LIN {X 0,Y 319.56,Z 711.312,A -85,B 0,C 180,E1 -15773.491,E2 -15773.491} C_VEL
LIN {X 0,Y 321.103,Z 700.055,A -85,B 0,C 180,E1 -15774.745,E2 -15774.745} C_VEL
LIN {X 0,Y 322.479,Z 688.391,A -85,B 0,C 180,E1 -15775.754,E2 -15775.754} C_VEL
LIN {X 0,Y 323.352,Z 677.795,A -85,B 0,C 180,E1 -15776.459,E2 -15776.459} C_VEL
LIN {X 0,Y 324.244,Z 665.597,A -85,B 0,C 180,E1 -15777.032,E2 -15777.032} C_VEL
LIN {X 0,Y 324.808,Z 650.654,A -85,B 0,C 180,E1 -15777.446,E2 -15777.446} C_VEL
LIN {X 0,Y 326.381,Z 586.086,A -85,B 0,C 180,E1 -15778.864,E2 -15778.864} C_VEL
LIN {X 0,Y 324.427,Z 577.286,A -85,B 0,C 180,E1 -15779.252,E2 -15779.252} C_VEL
LIN {X 0,Y 318.211,Z 562.488,A -85,B 0,C 180,E1 -15780.197,E2 -15780.197} C_VEL
LIN {X 0,Y 314.383,Z 553.731,A -85,B 0,C 180,E1 -15780.82,E2 -15780.82} C_VEL
LIN {X 0,Y 312.516,Z 545.559,A -85,B 0,C 180,E1 -15783.889,E2 -15783.889} C_VEL
LIN {X 0,Y 312.541,Z 545.551,A -85,B 0,C 180,E1 -15787.382,E2 -15787.382} C_VEL
LIN {X 0,Y 312.524,Z 545.556,A -85,B 0,C 180,E1 -15790.332,E2 -15790.332} C_VEL
LIN {X 0,Y 311.845,Z 545.642,A -85,B 0,C 180,E1 -15791.408,E2 -15791.408} C_VEL
LIN {X 0,Y 308.973,Z 545.997,A -85,B 0,C 180,E1 -15793.16,E2 -15793.16} C_VEL
LIN {X 0,Y 306.557,Z 546.301,A -85,B 0,C 180,E1 -15794.58,E2 -15794.58} C_VEL
LIN {X 0,Y 305.543,Z 546.423,A -85,B 0,C 180,E1 -15795.68,E2 -15795.68} C_VEL
LIN {X 0,Y 305.472,Z 546.432,A -85,B 0,C 180,E1 -15796.052,E2 -15796.052} C_VEL
LIN {X 0,Y 305.463,Z 546.425,A -85,B 0,C 180,E1 -15799.893,E2 -15799.893} C_VEL
LIN {X 0,Y 305.499,Z 546.428,A -85,B 0,C 180,E1 -15803.625,E2 -15803.625} C_VEL
LIN {X 0,Y 305.461,Z 546.432,A -85,B 0,C 180,E1 -15806.482,E2 -15806.482} C_VEL
LIN {X 0,Y 305.458,Z 546.428,A -85,B 0,C 180,E1 -15809.59,E2 -15809.59} C_VEL
LIN {X 0,Y 305.516,Z 546.425,A -85,B 0,C 180,E1 -15812.608,E2 -15812.608} C_VEL
LIN {X 0,Y 305.503,Z 546.429,A -85,B 0,C 180,E1 -15815.538,E2 -15815.538} C_VEL
LIN {X 0,Y 305.514,Z 546.427,A -85,B 0,C 180,E1 -15819.814,E2 -15819.814} C_VEL
LIN {X 0,Y 305.568,Z 546.415,A -85,B 0,C 180,E1 -15822.602,E2 -15822.602} C_VEL
LIN {X 0,Y 305.642,Z 546.411,A -85,B 0,C 180,E1 -15825.348,E2 -15825.348} C_VEL
LIN {X 0,Y 305.629,Z 546.413,A -85,B 0,C 180,E1 -15829.399,E2 -15829.399} C_VEL
LIN {X 0,Y 305.79,Z 546.386,A -85,B 0,C 180,E1 -15832.074,E2 -15832.074} C_VEL
LIN {X 0,Y 305.681,Z 546.41,A -85,B 0,C 180,E1 -15834.723,E2 -15834.723} C_VEL
LIN {X 0,Y 305.952,Z 546.367,A -85,B 0,C 180,E1 -15838.684,E2 -15838.684} C_VEL
LIN {X 0,Y 305.952,Z 546.372,A -85,B 0,C 180,E1 -15841.316,E2 -15841.316} C_VEL
LIN {X 0,Y 305.835,Z 546.389,A -85,B 0,C 180,E1 -15846.598,E2 -15846.598} C_VEL
LIN {X 0,Y 305.697,Z 546.4,A -85,B 0,C 180,E1 -15849.261,E2 -15849.261} C_VEL
LIN {X 0,Y 305.581,Z 546.409,A -85,B 0,C 180,E1 -15853.296,E2 -15853.296} C_VEL
LIN {X 0,Y 305.587,Z 546.419,A -85,B 0,C 180,E1 -15856.02,E2 -15856.02} C_VEL
LIN {X 0,Y 305.569,Z 546.418,A -85,B 0,C 180,E1 -15859.444,E2 -15859.444} C_VEL
LIN {X 0,Y 305.48,Z 546.426,A -85,B 0,C 180,E1 -15863.04,E2 -15863.04} C_VEL
LIN {X 0,Y 305.542,Z 546.423,A -85,B 0,C 180,E1 -15866.227,E2 -15866.227} C_VEL
LIN {X 0,Y 305.491,Z 546.431,A -85,B 0,C 180,E1 -15869.051,E2 -15869.051} C_VEL
LIN {X 0,Y 305.46,Z 546.434,A -85,B 0,C 180,E1 -15873.517,E2 -15873.517} C_VEL
LIN {X 0,Y 305.492,Z 546.434,A -85,B 0,C 180,E1 -15876.737,E2 -15876.737} C_VEL
LIN {X 0,Y 305.46,Z 546.438,A -85,B 0,C 180,E1 -15880.603,E2 -15880.603} C_VEL
LIN {X 0,Y 305.477,Z 546.434,A -85,B 0,C 180,E1 -15883.646,E2 -15883.646} C_VEL
LIN {X 0,Y 305.456,Z 546.437,A -85,B 0,C 180,E1 -15887.414,E2 -15887.414} C_VEL
LIN {X 0,Y 305.474,Z 546.435,A -85,B 0,C 180,E1 -15891.598,E2 -15891.598} C_VEL
LIN {X 0,Y 305.486,Z 546.463,A -85,B 0,C 180,E1 -15895.243,E2 -15895.243} C_VEL
LIN {X 0,Y 308.154,Z 557.631,A -85,B 0,C 180,E1 -15899.128,E2 -15899.128} C_VEL
LIN {X 0,Y 310.414,Z 568.645,A -85,B 0,C 180,E1 -15902.711,E2 -15902.711} C_VEL
LIN {X 0,Y 310.525,Z 569.174,A -85,B 0,C 180,E1 -15902.861,E2 -15902.861} C_VEL
LIN {X 0,Y 313.109,Z 576.135,A -85,B 0,C 180,E1 -15903.297,E2 -15903.297} C_VEL
LIN {X 0,Y 318.037,Z 602.027,A -85,B 0,C 180,E1 -15904.418,E2 -15904.418} C_VEL
LIN {X 0,Y 319.468,Z 612.293,A -85,B 0,C 180,E1 -15904.803,E2 -15904.803} C_VEL
LIN {X 0,Y 317.655,Z 677.964,A -85,B 0,C 180,E1 -15906.3,E2 -15906.3} C_VEL
LIN {X 0,Y 316.743,Z 691.271,A -85,B 0,C 180,E1 -15906.85,E2 -15906.85} C_VEL
LIN {X 0,Y 315.38,Z 704.306,A -85,B 0,C 180,E1 -15907.653,E2 -15907.653} C_VEL
LIN {X 0,Y 313.983,Z 716.101,A -85,B 0,C 180,E1 -15908.671,E2 -15908.671} C_VEL
LIN {X 0,Y 312.204,Z 727.465,A -85,B 0,C 180,E1 -15909.923,E2 -15909.923} C_VEL
LIN {X 0,Y 310.485,Z 737.722,A -85,B 0,C 180,E1 -15911.354,E2 -15911.354} C_VEL
LIN {X 0,Y 308.823,Z 747.523,A -85,B 0,C 180,E1 -15913.084,E2 -15913.084} C_VEL
LIN {X 0,Y 307.251,Z 756.594,A -85,B 0,C 180,E1 -15915.089,E2 -15915.089} C_VEL
LIN {X 0,Y 305.836,Z 763.695,A -85,B 0,C 180,E1 -15917.053,E2 -15917.053} C_VEL
LIN {X 0,Y 304.779,Z 770.182,A -85,B 0,C 180,E1 -15919.37,E2 -15919.37} C_VEL
LIN {X 0,Y 304.162,Z 774.48,A -85,B 0,C 180,E1 -15921.362,E2 -15921.362} C_VEL
LIN {X 0,Y 303.743,Z 777.719,A -85,B 0,C 180,E1 -15923.357,E2 -15923.357} C_VEL
LIN {X 0,Y 303.631,Z 780.557,A -85,B 0,C 180,E1 -15926.018,E2 -15926.018} C_VEL
LIN {X 0,Y 303.606,Z 781.339,A -85,B 0,C 180,E1 -15927.347,E2 -15927.347} C_VEL
LIN {X 0,Y 303.605,Z 781.714,A -85,B 0,C 180,E1 -15930,E2 -15930} C_VEL
LIN {X 0,Y 303.575,Z 781.323,A -85,B 0,C 180,E1 -15931.327,E2 -15931.327} C_VEL
LIN {X 0,Y 303.608,Z 780.508,A -85,B 0,C 180,E1 -15932.653,E2 -15932.653} C_VEL
LIN {X 0,Y 303.631,Z 779.27,A -85,B 0,C 180,E1 -15933.982,E2 -15933.982} C_VEL
LIN {X 0,Y 303.66,Z 777.217,A -85,B 0,C 180,E1 -15935.611,E2 -15935.611} C_VEL
LIN {X 0,Y 303.953,Z 772.983,A -85,B 0,C 180,E1 -15937.974,E2 -15937.974} C_VEL
LIN {X 0,Y 304.414,Z 768.207,A -85,B 0,C 180,E1 -15939.971,E2 -15939.971} C_VEL
LIN {X 0,Y 305.31,Z 761.043,A -85,B 0,C 180,E1 -15942.294,E2 -15942.294} C_VEL
LIN {X 0,Y 306.496,Z 753.237,A -85,B 0,C 180,E1 -15944.27,E2 -15944.27} C_VEL
LIN {X 0,Y 307.813,Z 743.859,A -85,B 0,C 180,E1 -15946.165,E2 -15946.165} C_VEL
LIN {X 0,Y 309.152,Z 733.316,A -85,B 0,C 180,E1 -15947.872,E2 -15947.872} C_VEL
LIN {X 0,Y 310.628,Z 721.827,A -85,B 0,C 180,E1 -15949.322,E2 -15949.322} C_VEL
LIN {X 0,Y 311.964,Z 710.545,A -85,B 0,C 180,E1 -15950.437,E2 -15950.437} C_VEL
LIN {X 0,Y 313.093,Z 699.088,A -85,B 0,C 180,E1 -15951.306,E2 -15951.306} C_VEL
LIN {X 0,Y 314.068,Z 685.985,A -85,B 0,C 180,E1 -15952.013,E2 -15952.013} C_VEL
LIN {X 0,Y 314.673,Z 672.398,A -85,B 0,C 180,E1 -15952.472,E2 -15952.472} C_VEL
LIN {X 0,Y 316.012,Z 609.471,A -85,B 0,C 180,E1 -15953.888,E2 -15953.888} C_VEL
LIN {X 0,Y 311.128,Z 577.16,A -85,B 0,C 180,E1 -15955.044,E2 -15955.044} C_VEL
LIN {X 0,Y 309.749,Z 569.178,A -85,B 0,C 180,E1 -15955.394,E2 -15955.394} C_VEL
LIN {X 0,Y 309.315,Z 564.88,A -85,B 0,C 180,E1 -15956.662,E2 -15956.662} C_VEL
LIN {X 0,Y 307.408,Z 555.133,A -85,B 0,C 180,E1 -15959.685,E2 -15959.685} C_VEL
LIN {X 0,Y 305.487,Z 546.434,A -85,B 0,C 180,E1 -15962.531,E2 -15962.531} C_VEL
LIN {X 0,Y 305.494,Z 546.43,A -85,B 0,C 180,E1 -15966.736,E2 -15966.736} C_VEL
LIN {X 0,Y 305.452,Z 546.434,A -85,B 0,C 180,E1 -15970.599,E2 -15970.599} C_VEL
LIN {X 0,Y 305.424,Z 546.437,A -85,B 0,C 180,E1 -15974.493,E2 -15974.493} C_VEL
LIN {X 0,Y 305.475,Z 546.432,A -85,B 0,C 180,E1 -15978.149,E2 -15978.149} C_VEL
LIN {X 0,Y 305.504,Z 546.431,A -85,B 0,C 180,E1 -15981.602,E2 -15981.602} C_VEL
LIN {X 0,Y 305.457,Z 546.434,A -85,B 0,C 180,E1 -15984.886,E2 -15984.886} C_VEL
LIN {X 0,Y 305.446,Z 546.434,A -85,B 0,C 180,E1 -15988.355,E2 -15988.355} C_VEL
LIN {X 0,Y 305.515,Z 546.428,A -85,B 0,C 180,E1 -15991.113,E2 -15991.113} C_VEL
LIN {X 0,Y 305.565,Z 546.42,A -85,B 0,C 180,E1 -15994.087,E2 -15994.087} C_VEL
LIN {X 0,Y 305.475,Z 546.43,A -85,B 0,C 180,E1 -15998.401,E2 -15998.401} C_VEL
LIN {X 0,Y 305.573,Z 546.422,A -85,B 0,C 180,E1 -16001.217,E2 -16001.217} C_VEL
LIN {X 0,Y 305.642,Z 546.414,A -85,B 0,C 180,E1 -16005.349,E2 -16005.349} C_VEL
LIN {X 0,Y 305.631,Z 546.412,A -85,B 0,C 180,E1 -16009.4,E2 -16009.4} C_VEL
LIN {X 0,Y 305.802,Z 546.391,A -85,B 0,C 180,E1 -16012.074,E2 -16012.074} C_VEL
LIN {X 0,Y 305.681,Z 546.403,A -85,B 0,C 180,E1 -16014.723,E2 -16014.723} C_VEL
LIN {X 0,Y 305.95,Z 546.372,A -85,B 0,C 180,E1 -16018.684,E2 -16018.684} C_VEL
LIN {X 0,Y 305.95,Z 546.374,A -85,B 0,C 180,E1 -16021.316,E2 -16021.316} C_VEL
LIN {X 0,Y 305.682,Z 546.408,A -85,B 0,C 180,E1 -16025.277,E2 -16025.277} C_VEL
LIN {X 0,Y 305.79,Z 546.391,A -85,B 0,C 180,E1 -16027.926,E2 -16027.926} C_VEL
LIN {X 0,Y 305.596,Z 546.413,A -85,B 0,C 180,E1 -16031.946,E2 -16031.946} C_VEL
LIN {X 0,Y 305.631,Z 546.413,A -85,B 0,C 180,E1 -16035.035,E2 -16035.035} C_VEL
LIN {X 0,Y 305.57,Z 546.417,A -85,B 0,C 180,E1 -16039.445,E2 -16039.445} C_VEL
LIN {X 0,Y 305.485,Z 546.431,A -85,B 0,C 180,E1 -16043.042,E2 -16043.042} C_VEL
LIN {X 0,Y 305.543,Z 546.421,A -85,B 0,C 180,E1 -16046.228,E2 -16046.228} C_VEL
LIN {X 0,Y 305.491,Z 546.431,A -85,B 0,C 180,E1 -16049.051,E2 -16049.051} C_VEL
LIN {X 0,Y 305.461,Z 546.437,A -85,B 0,C 180,E1 -16053.518,E2 -16053.518} C_VEL
LIN {X 0,Y 305.493,Z 546.426,A -85,B 0,C 180,E1 -16056.737,E2 -16056.737} C_VEL
LIN {X 0,Y 305.452,Z 546.434,A -85,B 0,C 180,E1 -16060.601,E2 -16060.601} C_VEL
LIN {X 0,Y 305.468,Z 546.435,A -85,B 0,C 180,E1 -16063.648,E2 -16063.648} C_VEL
LIN {X 0,Y 305.507,Z 546.432,A -85,B 0,C 180,E1 -16067.404,E2 -16067.404} C_VEL
LIN {X 0,Y 305.519,Z 546.429,A -85,B 0,C 180,E1 -16071.605,E2 -16071.605} C_VEL
LIN {X 0,Y 305.462,Z 546.434,A -85,B 0,C 180,E1 -16074.888,E2 -16074.888} C_VEL
LIN {X 0,Y 305.452,Z 546.435,A -85,B 0,C 180,E1 -16078.356,E2 -16078.356} C_VEL
LIN {X 0,Y 305.521,Z 546.431,A -85,B 0,C 180,E1 -16081.115,E2 -16081.115} C_VEL
LIN {X 0,Y 305.574,Z 546.419,A -85,B 0,C 180,E1 -16084.089,E2 -16084.089} C_VEL
LIN {X 0,Y 305.566,Z 546.631,A -85,B 0,C 180,E1 -16085.98,E2 -16085.98} C_VEL
LIN {X 0,Y 307.028,Z 553.759,A -85,B 0,C 180,E1 -16088.494,E2 -16088.494} C_VEL
LIN {X 0,Y 314.277,Z 572.979,A -85,B 0,C 180,E1 -16089.556,E2 -16089.556} C_VEL
LIN {X 0,Y 316.555,Z 584.974,A -85,B 0,C 180,E1 -16090.02,E2 -16090.02} C_VEL
LIN {X 0,Y 314.853,Z 660.952,A -85,B 0,C 180,E1 -16091.757,E2 -16091.757} C_VEL
LIN {X 0,Y 314.205,Z 673.84,A -85,B 0,C 180,E1 -16092.299,E2 -16092.299} C_VEL
LIN {X 0,Y 313.3,Z 685.911,A -85,B 0,C 180,E1 -16093.046,E2 -16093.046} C_VEL
LIN {X 0,Y 312.168,Z 697.305,A -85,B 0,C 180,E1 -16093.991,E2 -16093.991} C_VEL
LIN {X 0,Y 310.905,Z 708.975,A -85,B 0,C 180,E1 -16095.268,E2 -16095.268} C_VEL
LIN {X 0,Y 309.493,Z 719.45,A -85,B 0,C 180,E1 -16096.708,E2 -16096.708} C_VEL
LIN {X 0,Y 308.138,Z 728.021,A -85,B 0,C 180,E1 -16098.155,E2 -16098.155} C_VEL
LIN {X 0,Y 307.155,Z 735.978,A -85,B 0,C 180,E1 -16099.805,E2 -16099.805} C_VEL
LIN {X 0,Y 306.074,Z 743.623,A -85,B 0,C 180,E1 -16101.749,E2 -16101.749} C_VEL
LIN {X 0,Y 305.32,Z 748.885,A -85,B 0,C 180,E1 -16103.391,E2 -16103.391} C_VEL
LIN {X 0,Y 304.67,Z 754.01,A -85,B 0,C 180,E1 -16105.369,E2 -16105.369} C_VEL
LIN {X 0,Y 303.991,Z 758.003,A -85,B 0,C 180,E1 -16107.35,E2 -16107.35} C_VEL
LIN {X 0,Y 303.805,Z 760.064,A -85,B 0,C 180,E1 -16108.674,E2 -16108.674} C_VEL
LIN {X 0,Y 303.616,Z 762.942,A -85,B 0,C 180,E1 -16111.326,E2 -16111.326} C_VEL
LIN {X 0,Y 303.632,Z 763.785,A -85,B 0,C 180,E1 -16112.653,E2 -16112.653} C_VEL
LIN {X 0,Y 303.647,Z 764.2,A -85,B 0,C 180,E1 -16113.981,E2 -16113.981} C_VEL
LIN {X 0,Y 303.697,Z 764.191,A -85,B 0,C 180,E1 -16115.678,E2 -16115.678} C_VEL
LIN {X 0,Y 303.777,Z 763.154,A -85,B 0,C 180,E1 -16117.979,E2 -16117.979} C_VEL
LIN {X 0,Y 303.939,Z 761.978,A -85,B 0,C 180,E1 -16119.315,E2 -16119.315} C_VEL
LIN {X 0,Y 304.161,Z 760.397,A -85,B 0,C 180,E1 -16120.652,E2 -16120.652} C_VEL
LIN {X 0,Y 304.752,Z 757.208,A -85,B 0,C 180,E1 -16122.655,E2 -16122.655} C_VEL
LIN {X 0,Y 305.742,Z 751.858,A -85,B 0,C 180,E1 -16125.105,E2 -16125.105} C_VEL
LIN {X 0,Y 306.938,Z 745.372,A -85,B 0,C 180,E1 -16127.317,E2 -16127.317} C_VEL
LIN {X 0,Y 308.349,Z 737.987,A -85,B 0,C 180,E1 -16129.298,E2 -16129.298} C_VEL
LIN {X 0,Y 309.874,Z 730.443,A -85,B 0,C 180,E1 -16130.929,E2 -16130.929} C_VEL
LIN {X 0,Y 311.396,Z 721.288,A -85,B 0,C 180,E1 -16132.561,E2 -16132.561} C_VEL
LIN {X 0,Y 313.002,Z 711.086,A -85,B 0,C 180,E1 -16134.014,E2 -16134.014} C_VEL
LIN {X 0,Y 314.624,Z 699.733,A -85,B 0,C 180,E1 -16135.29,E2 -16135.29} C_VEL
LIN {X 0,Y 316.05,Z 687.935,A -85,B 0,C 180,E1 -16136.317,E2 -16136.317} C_VEL
LIN {X 0,Y 316.984,Z 677.136,A -85,B 0,C 180,E1 -16137.033,E2 -16137.033} C_VEL
LIN {X 0,Y 317.861,Z 664.324,A -85,B 0,C 180,E1 -16137.621,E2 -16137.621} C_VEL
LIN {X 0,Y 318.495,Z 646.755,A -85,B 0,C 180,E1 -16138.08,E2 -16138.08} C_VEL
LIN {X 0,Y 319.984,Z 586.641,A -85,B 0,C 180,E1 -16139.429,E2 -16139.429} C_VEL
LIN {X 0,Y 318.28,Z 579.564,A -85,B 0,C 180,E1 -16139.764,E2 -16139.764} C_VEL
LIN {X 0,Y 311.901,Z 564.373,A -85,B 0,C 180,E1 -16140.769,E2 -16140.769} C_VEL
LIN {X 0,Y 307.227,Z 553.981,A -85,B 0,C 180,E1 -16141.541,E2 -16141.541} C_VEL
LIN {X 0,Y 305.461,Z 546.438,A -85,B 0,C 180,E1 -16144.464,E2 -16144.464} C_VEL
LIN {X 0,Y 305.509,Z 546.427,A -85,B 0,C 180,E1 -16148.396,E2 -16148.396} C_VEL
LIN {X 0,Y 305.507,Z 546.432,A -85,B 0,C 180,E1 -16152.596,E2 -16152.596} C_VEL
LIN {X 0,Y 305.472,Z 546.432,A -85,B 0,C 180,E1 -16156.052,E2 -16156.052} C_VEL
LIN {X 0,Y 304.825,Z 546.516,A -85,B 0,C 180,E1 -16157.152,E2 -16157.152} C_VEL
LIN {X 0,Y 301.953,Z 546.873,A -85,B 0,C 180,E1 -16158.94,E2 -16158.94} C_VEL
LIN {X 0,Y 299.517,Z 547.173,A -85,B 0,C 180,E1 -16160.392,E2 -16160.392} C_VEL
LIN {X 0,Y 298.495,Z 547.303,A -85,B 0,C 180,E1 -16161.517,E2 -16161.517} C_VEL
LIN {X 0,Y 298.425,Z 547.31,A -85,B 0,C 180,E1 -16161.898,E2 -16161.898} C_VEL
LIN {X 0,Y 298.404,Z 547.311,A -85,B 0,C 180,E1 -16165.58,E2 -16165.58} C_VEL
LIN {X 0,Y 298.391,Z 547.313,A -85,B 0,C 180,E1 -16168.79,E2 -16168.79} C_VEL
LIN {X 0,Y 298.459,Z 547.307,A -85,B 0,C 180,E1 -16171.904,E2 -16171.904} C_VEL
LIN {X 0,Y 298.48,Z 547.306,A -85,B 0,C 180,E1 -16174.923,E2 -16174.923} C_VEL
LIN {X 0,Y 298.445,Z 547.309,A -85,B 0,C 180,E1 -16179.315,E2 -16179.315} C_VEL
LIN {X 0,Y 298.531,Z 547.291,A -85,B 0,C 180,E1 -16182.179,E2 -16182.179} C_VEL
LIN {X 0,Y 298.587,Z 547.291,A -85,B 0,C 180,E1 -16184.994,E2 -16184.994} C_VEL
LIN {X 0,Y 298.585,Z 547.292,A -85,B 0,C 180,E1 -16189.146,E2 -16189.146} C_VEL
LIN {X 0,Y 298.734,Z 547.266,A -85,B 0,C 180,E1 -16191.885,E2 -16191.885} C_VEL
LIN {X 0,Y 298.652,Z 547.284,A -85,B 0,C 180,E1 -16194.599,E2 -16194.599} C_VEL
LIN {X 0,Y 298.918,Z 547.242,A -85,B 0,C 180,E1 -16198.653,E2 -16198.653} C_VEL
LIN {X 0,Y 298.918,Z 547.248,A -85,B 0,C 180,E1 -16201.347,E2 -16201.347} C_VEL
LIN {X 0,Y 298.78,Z 547.266,A -85,B 0,C 180,E1 -16206.754,E2 -16206.754} C_VEL
LIN {X 0,Y 298.629,Z 547.281,A -85,B 0,C 180,E1 -16209.482,E2 -16209.482} C_VEL
LIN {X 0,Y 298.545,Z 547.285,A -85,B 0,C 180,E1 -16213.616,E2 -16213.616} C_VEL
LIN {X 0,Y 298.542,Z 547.299,A -85,B 0,C 180,E1 -16216.409,E2 -16216.409} C_VEL
LIN {X 0,Y 298.504,Z 547.298,A -85,B 0,C 180,E1 -16219.654,E2 -16219.654} C_VEL
LIN {X 0,Y 298.423,Z 547.306,A -85,B 0,C 180,E1 -16223.601,E2 -16223.601} C_VEL
LIN {X 0,Y 298.484,Z 547.299,A -85,B 0,C 180,E1 -16226.575,E2 -16226.575} C_VEL
LIN {X 0,Y 298.416,Z 547.311,A -85,B 0,C 180,E1 -16229.641,E2 -16229.641} C_VEL
LIN {X 0,Y 298.39,Z 547.317,A -85,B 0,C 180,E1 -16232.801,E2 -16232.801} C_VEL
LIN {X 0,Y 298.461,Z 547.309,A -85,B 0,C 180,E1 -16236.813,E2 -16236.813} C_VEL
LIN {X 0,Y 298.415,Z 547.314,A -85,B 0,C 180,E1 -16241.095,E2 -16241.095} C_VEL
LIN {X 0,Y 298.385,Z 547.319,A -85,B 0,C 180,E1 -16244.959,E2 -16244.959} C_VEL
LIN {X 0,Y 298.385,Z 547.319,A -85,B 0,C 180,E1 -16248.913,E2 -16248.913} C_VEL
LIN {X 0,Y 298.444,Z 547.31,A -85,B 0,C 180,E1 -16253.193,E2 -16253.193} C_VEL
LIN {X 0,Y 298.467,Z 547.491,A -85,B 0,C 180,E1 -16254.661,E2 -16254.661} C_VEL
LIN {X 0,Y 301.166,Z 558.807,A -85,B 0,C 180,E1 -16258.721,E2 -16258.721} C_VEL
LIN {X 0,Y 303.324,Z 569.024,A -85,B 0,C 180,E1 -16262.11,E2 -16262.11} C_VEL
LIN {X 0,Y 307.136,Z 578.741,A -85,B 0,C 180,E1 -16262.765,E2 -16262.765} C_VEL
LIN {X 0,Y 311.765,Z 603.378,A -85,B 0,C 180,E1 -16263.861,E2 -16263.861} C_VEL
LIN {X 0,Y 313.119,Z 613.122,A -85,B 0,C 180,E1 -16264.238,E2 -16264.238} C_VEL
LIN {X 0,Y 311.298,Z 677.056,A -85,B 0,C 180,E1 -16265.715,E2 -16265.715} C_VEL
LIN {X 0,Y 310.396,Z 690.278,A -85,B 0,C 180,E1 -16266.26,E2 -16266.26} C_VEL
LIN {X 0,Y 309.097,Z 702.433,A -85,B 0,C 180,E1 -16266.997,E2 -16266.997} C_VEL
LIN {X 0,Y 307.628,Z 714.698,A -85,B 0,C 180,E1 -16268.032,E2 -16268.032} C_VEL
LIN {X 0,Y 305.781,Z 726.28,A -85,B 0,C 180,E1 -16269.307,E2 -16269.307} C_VEL
LIN {X 0,Y 303.959,Z 736.711,A -85,B 0,C 180,E1 -16270.763,E2 -16270.763} C_VEL
LIN {X 0,Y 302.138,Z 746.571,A -85,B 0,C 180,E1 -16272.496,E2 -16272.496} C_VEL
LIN {X 0,Y 300.619,Z 755.195,A -85,B 0,C 180,E1 -16274.404,E2 -16274.404} C_VEL
LIN {X 0,Y 299.147,Z 762.523,A -85,B 0,C 180,E1 -16276.413,E2 -16276.413} C_VEL
LIN {X 0,Y 298.083,Z 768.412,A -85,B 0,C 180,E1 -16278.44,E2 -16278.44} C_VEL
LIN {X 0,Y 297.302,Z 773.065,A -85,B 0,C 180,E1 -16280.475,E2 -16280.475} C_VEL
LIN {X 0,Y 296.804,Z 776.619,A -85,B 0,C 180,E1 -16282.517,E2 -16282.517} C_VEL
LIN {X 0,Y 296.552,Z 779.176,A -85,B 0,C 180,E1 -16284.561,E2 -16284.561} C_VEL
LIN {X 0,Y 296.528,Z 780.382,A -85,B 0,C 180,E1 -16285.923,E2 -16285.923} C_VEL
LIN {X 0,Y 296.533,Z 781.148,A -85,B 0,C 180,E1 -16287.283,E2 -16287.283} C_VEL
LIN {X 0,Y 296.52,Z 781.505,A -85,B 0,C 180,E1 -16290,E2 -16290} C_VEL
LIN {X 0,Y 296.494,Z 781.104,A -85,B 0,C 180,E1 -16291.358,E2 -16291.358} C_VEL
LIN {X 0,Y 296.534,Z 780.27,A -85,B 0,C 180,E1 -16292.717,E2 -16292.717} C_VEL
LIN {X 0,Y 296.529,Z 779.022,A -85,B 0,C 180,E1 -16294.077,E2 -16294.077} C_VEL
LIN {X 0,Y 296.553,Z 777.257,A -85,B 0,C 180,E1 -16295.522,E2 -16295.522} C_VEL
LIN {X 0,Y 296.786,Z 774.037,A -85,B 0,C 180,E1 -16297.483,E2 -16297.483} C_VEL
LIN {X 0,Y 297.214,Z 769.628,A -85,B 0,C 180,E1 -16299.527,E2 -16299.527} C_VEL
LIN {X 0,Y 297.873,Z 764.015,A -85,B 0,C 180,E1 -16301.569,E2 -16301.569} C_VEL
LIN {X 0,Y 298.899,Z 757.005,A -85,B 0,C 180,E1 -16303.599,E2 -16303.599} C_VEL
LIN {X 0,Y 300.253,Z 748.214,A -85,B 0,C 180,E1 -16305.615,E2 -16305.615} C_VEL
LIN {X 0,Y 301.512,Z 739.161,A -85,B 0,C 180,E1 -16307.296,E2 -16307.296} C_VEL
LIN {X 0,Y 302.862,Z 729.288,A -85,B 0,C 180,E1 -16308.782,E2 -16308.782} C_VEL
LIN {X 0,Y 304.321,Z 718.323,A -85,B 0,C 180,E1 -16310.091,E2 -16310.091} C_VEL
LIN {X 0,Y 305.682,Z 706.008,A -85,B 0,C 180,E1 -16311.229,E2 -16311.229} C_VEL
LIN {X 0,Y 306.896,Z 693.027,A -85,B 0,C 180,E1 -16312.112,E2 -16312.112} C_VEL
LIN {X 0,Y 307.767,Z 679.818,A -85,B 0,C 180,E1 -16312.709,E2 -16312.709} C_VEL
LIN {X 0,Y 308.395,Z 658.837,A -85,B 0,C 180,E1 -16313.246,E2 -16313.246} C_VEL
LIN {X 0,Y 309.372,Z 609.883,A -85,B 0,C 180,E1 -16314.375,E2 -16314.375} C_VEL
LIN {X 0,Y 304.698,Z 578.701,A -85,B 0,C 180,E1 -16315.522,E2 -16315.522} C_VEL
LIN {X 0,Y 302.837,Z 569.074,A -85,B 0,C 180,E1 -16315.936,E2 -16315.936} C_VEL
LIN {X 0,Y 301.088,Z 559.401,A -85,B 0,C 180,E1 -16318.969,E2 -16318.969} C_VEL
LIN {X 0,Y 298.936,Z 549.638,A -85,B 0,C 180,E1 -16322.182,E2 -16322.182} C_VEL
LIN {X 0,Y 298.426,Z 547.314,A -85,B 0,C 180,E1 -16322.996,E2 -16322.996} C_VEL
LIN {X 0,Y 298.463,Z 547.306,A -85,B 0,C 180,E1 -16326.812,E2 -16326.812} C_VEL
LIN {X 0,Y 298.385,Z 547.317,A -85,B 0,C 180,E1 -16331.087,E2 -16331.087} C_VEL
LIN {X 0,Y 298.385,Z 547.316,A -85,B 0,C 180,E1 -16335.041,E2 -16335.041} C_VEL
LIN {X 0,Y 298.415,Z 547.312,A -85,B 0,C 180,E1 -16338.905,E2 -16338.905} C_VEL
LIN {X 0,Y 298.461,Z 547.307,A -85,B 0,C 180,E1 -16343.187,E2 -16343.187} C_VEL
LIN {X 0,Y 298.39,Z 547.315,A -85,B 0,C 180,E1 -16347.199,E2 -16347.199} C_VEL
LIN {X 0,Y 298.427,Z 547.309,A -85,B 0,C 180,E1 -16350.614,E2 -16350.614} C_VEL
LIN {X 0,Y 298.478,Z 547.306,A -85,B 0,C 180,E1 -16353.474,E2 -16353.474} C_VEL
LIN {X 0,Y 298.425,Z 547.307,A -85,B 0,C 180,E1 -16356.699,E2 -16356.699} C_VEL
LIN {X 0,Y 298.519,Z 547.298,A -85,B 0,C 180,E1 -16360.756,E2 -16360.756} C_VEL
LIN {X 0,Y 298.587,Z 547.29,A -85,B 0,C 180,E1 -16364.995,E2 -16364.995} C_VEL
LIN {X 0,Y 298.586,Z 547.288,A -85,B 0,C 180,E1 -16369.146,E2 -16369.146} C_VEL
LIN {X 0,Y 298.748,Z 547.271,A -85,B 0,C 180,E1 -16371.886,E2 -16371.886} C_VEL
LIN {X 0,Y 298.652,Z 547.278,A -85,B 0,C 180,E1 -16374.599,E2 -16374.599} C_VEL
LIN {X 0,Y 298.916,Z 547.248,A -85,B 0,C 180,E1 -16378.653,E2 -16378.653} C_VEL
LIN {X 0,Y 298.916,Z 547.249,A -85,B 0,C 180,E1 -16381.347,E2 -16381.347} C_VEL
LIN {X 0,Y 298.781,Z 547.265,A -85,B 0,C 180,E1 -16386.754,E2 -16386.754} C_VEL
LIN {X 0,Y 298.628,Z 547.281,A -85,B 0,C 180,E1 -16389.482,E2 -16389.482} C_VEL
LIN {X 0,Y 298.545,Z 547.297,A -85,B 0,C 180,E1 -16393.616,E2 -16393.616} C_VEL
LIN {X 0,Y 298.543,Z 547.294,A -85,B 0,C 180,E1 -16396.409,E2 -16396.409} C_VEL
LIN {X 0,Y 298.505,Z 547.295,A -85,B 0,C 180,E1 -16399.655,E2 -16399.655} C_VEL
LIN {X 0,Y 298.452,Z 547.31,A -85,B 0,C 180,E1 -16403.598,E2 -16403.598} C_VEL
LIN {X 0,Y 298.485,Z 547.3,A -85,B 0,C 180,E1 -16406.575,E2 -16406.575} C_VEL
LIN {X 0,Y 298.416,Z 547.313,A -85,B 0,C 180,E1 -16409.642,E2 -16409.642} C_VEL
LIN {X 0,Y 298.392,Z 547.313,A -85,B 0,C 180,E1 -16412.801,E2 -16412.801} C_VEL
LIN {X 0,Y 298.461,Z 547.302,A -85,B 0,C 180,E1 -16416.813,E2 -16416.813} C_VEL
LIN {X 0,Y 298.41,Z 547.315,A -85,B 0,C 180,E1 -16421.258,E2 -16421.258} C_VEL
LIN {X 0,Y 298.415,Z 547.313,A -85,B 0,C 180,E1 -16425.048,E2 -16425.048} C_VEL
LIN {X 0,Y 298.45,Z 547.306,A -85,B 0,C 180,E1 -16428.751,E2 -16428.751} C_VEL
LIN {X 0,Y 298.47,Z 547.307,A -85,B 0,C 180,E1 -16433.187,E2 -16433.187} C_VEL
LIN {X 0,Y 298.395,Z 547.317,A -85,B 0,C 180,E1 -16437.201,E2 -16437.201} C_VEL
LIN {X 0,Y 298.471,Z 547.308,A -85,B 0,C 180,E1 -16441.906,E2 -16441.906} C_VEL
LIN {X 0,Y 298.48,Z 547.348,A -85,B 0,C 180,E1 -16445.482,E2 -16445.482} C_VEL
LIN {X 0,Y 299.861,Z 553.96,A -85,B 0,C 180,E1 -16447.886,E2 -16447.886} C_VEL
LIN {X 0,Y 307.981,Z 575.178,A -85,B 0,C 180,E1 -16449.113,E2 -16449.113} C_VEL
LIN {X 0,Y 309.97,Z 586.458,A -85,B 0,C 180,E1 -16449.551,E2 -16449.551} C_VEL
LIN {X 0,Y 308.241,Z 660.816,A -85,B 0,C 180,E1 -16451.282,E2 -16451.282} C_VEL
LIN {X 0,Y 307.595,Z 673.526,A -85,B 0,C 180,E1 -16451.819,E2 -16451.819} C_VEL
LIN {X 0,Y 306.667,Z 685.73,A -85,B 0,C 180,E1 -16452.581,E2 -16452.581} C_VEL
LIN {X 0,Y 305.389,Z 698.049,A -85,B 0,C 180,E1 -16453.626,E2 -16453.626} C_VEL
LIN {X 0,Y 304.085,Z 709.602,A -85,B 0,C 180,E1 -16454.93,E2 -16454.93} C_VEL
LIN {X 0,Y 302.634,Z 720.004,A -85,B 0,C 180,E1 -16456.401,E2 -16456.401} C_VEL
LIN {X 0,Y 301.217,Z 728.519,A -85,B 0,C 180,E1 -16457.879,E2 -16457.879} C_VEL
LIN {X 0,Y 300.187,Z 736.427,A -85,B 0,C 180,E1 -16459.565,E2 -16459.565} C_VEL
LIN {X 0,Y 299.088,Z 744.01,A -85,B 0,C 180,E1 -16461.555,E2 -16461.555} C_VEL
LIN {X 0,Y 298.022,Z 751.058,A -85,B 0,C 180,E1 -16463.908,E2 -16463.908} C_VEL
LIN {X 0,Y 297.241,Z 755.764,A -85,B 0,C 180,E1 -16465.933,E2 -16465.933} C_VEL
LIN {X 0,Y 296.926,Z 759.361,A -85,B 0,C 180,E1 -16467.965,E2 -16467.965} C_VEL
LIN {X 0,Y 296.583,Z 761.966,A -85,B 0,C 180,E1 -16470,E2 -16470} C_VEL
LIN {X 0,Y 296.533,Z 763.193,A -85,B 0,C 180,E1 -16471.358,E2 -16471.358} C_VEL
LIN {X 0,Y 296.557,Z 764.012,A -85,B 0,C 180,E1 -16472.717,E2 -16472.717} C_VEL
LIN {X 0,Y 296.562,Z 764.411,A -85,B 0,C 180,E1 -16474.077,E2 -16474.077} C_VEL
LIN {X 0,Y 296.582,Z 764.417,A -85,B 0,C 180,E1 -16475.577,E2 -16475.577} C_VEL
LIN {X 0,Y 296.7,Z 763.318,A -85,B 0,C 180,E1 -16478.171,E2 -16478.171} C_VEL
LIN {X 0,Y 296.89,Z 762.124,A -85,B 0,C 180,E1 -16479.538,E2 -16479.538} C_VEL
LIN {X 0,Y 297.318,Z 759.577,A -85,B 0,C 180,E1 -16481.591,E2 -16481.591} C_VEL
LIN {X 0,Y 297.989,Z 756.018,A -85,B 0,C 180,E1 -16483.641,E2 -16483.641} C_VEL
LIN {X 0,Y 298.907,Z 751.501,A -85,B 0,C 180,E1 -16485.624,E2 -16485.624} C_VEL
LIN {X 0,Y 300.103,Z 745.392,A -85,B 0,C 180,E1 -16487.724,E2 -16487.724} C_VEL
LIN {X 0,Y 301.609,Z 737.968,A -85,B 0,C 180,E1 -16489.747,E2 -16489.747} C_VEL
LIN {X 0,Y 303.172,Z 730.379,A -85,B 0,C 180,E1 -16491.414,E2 -16491.414} C_VEL
LIN {X 0,Y 304.767,Z 721.161,A -85,B 0,C 180,E1 -16493.08,E2 -16493.08} C_VEL
LIN {X 0,Y 306.482,Z 710.863,A -85,B 0,C 180,E1 -16494.558,E2 -16494.558} C_VEL
LIN {X 0,Y 308.205,Z 699.416,A -85,B 0,C 180,E1 -16495.855,E2 -16495.855} C_VEL
LIN {X 0,Y 309.658,Z 687.461,A -85,B 0,C 180,E1 -16496.904,E2 -16496.904} C_VEL
LIN {X 0,Y 310.655,Z 676.413,A -85,B 0,C 180,E1 -16497.63,E2 -16497.63} C_VEL
LIN {X 0,Y 311.547,Z 663.017,A -85,B 0,C 180,E1 -16498.23,E2 -16498.23} C_VEL
LIN {X 0,Y 312.344,Z 639.755,A -85,B 0,C 180,E1 -16498.807,E2 -16498.807} C_VEL
LIN {X 0,Y 313.662,Z 587.865,A -85,B 0,C 180,E1 -16499.995,E2 -16499.995} C_VEL
LIN {X 0,Y 312.287,Z 582.261,A -85,B 0,C 180,E1 -16500.272,E2 -16500.272} C_VEL
LIN {X 0,Y 307.035,Z 569.589,A -85,B 0,C 180,E1 -16501.129,E2 -16501.129} C_VEL
LIN {X 0,Y 300.007,Z 554.267,A -85,B 0,C 180,E1 -16502.294,E2 -16502.294} C_VEL
LIN {X 0,Y 298.428,Z 547.31,A -85,B 0,C 180,E1 -16505.03,E2 -16505.03} C_VEL
LIN {X 0,Y 298.44,Z 547.306,A -85,B 0,C 180,E1 -16507.753,E2 -16507.753} C_VEL
LIN {X 0,Y 298.451,Z 547.308,A -85,B 0,C 180,E1 -16511.249,E2 -16511.249} C_VEL
LIN {X 0,Y 298.415,Z 547.312,A -85,B 0,C 180,E1 -16515.046,E2 -16515.046} C_VEL
LIN {X 0,Y 298.418,Z 547.298,A -85,B 0,C 180,E1 -16518.743,E2 -16518.743} C_VEL
LIN {X 0,Y 298.425,Z 547.31,A -85,B 0,C 180,E1 -16521.898,E2 -16521.898} C_VEL
LIN {X 0,Y 297.773,Z 547.394,A -85,B 0,C 180,E1 -16523.024,E2 -16523.024} C_VEL
LIN {X 0,Y 294.862,Z 547.757,A -85,B 0,C 180,E1 -16524.856,E2 -16524.856} C_VEL
LIN {X 0,Y 292.413,Z 548.06,A -85,B 0,C 180,E1 -16526.344,E2 -16526.344} C_VEL
LIN {X 0,Y 291.414,Z 548.185,A -85,B 0,C 180,E1 -16527.498,E2 -16527.498} C_VEL
LIN {X 0,Y 291.362,Z 548.191,A -85,B 0,C 180,E1 -16527.888,E2 -16527.888} C_VEL
LIN {X 0,Y 291.378,Z 548.19,A -85,B 0,C 180,E1 -16531.158,E2 -16531.158} C_VEL
LIN {X 0,Y 291.411,Z 548.179,A -85,B 0,C 180,E1 -16534.271,E2 -16534.271} C_VEL
LIN {X 0,Y 291.376,Z 548.181,A -85,B 0,C 180,E1 -16537.299,E2 -16537.299} C_VEL
LIN {X 0,Y 291.453,Z 548.181,A -85,B 0,C 180,E1 -16540.27,E2 -16540.27} C_VEL
LIN {X 0,Y 291.55,Z 548.17,A -85,B 0,C 180,E1 -16544.623,E2 -16544.623} C_VEL
LIN {X 0,Y 291.529,Z 548.17,A -85,B 0,C 180,E1 -16548.88,E2 -16548.88} C_VEL
LIN {X 0,Y 291.681,Z 548.145,A -85,B 0,C 180,E1 -16551.687,E2 -16551.687} C_VEL
LIN {X 0,Y 291.622,Z 548.158,A -85,B 0,C 180,E1 -16554.468,E2 -16554.468} C_VEL
LIN {X 0,Y 291.884,Z 548.118,A -85,B 0,C 180,E1 -16558.62,E2 -16558.62} C_VEL
LIN {X 0,Y 291.884,Z 548.124,A -85,B 0,C 180,E1 -16561.38,E2 -16561.38} C_VEL
LIN {X 0,Y 291.729,Z 548.143,A -85,B 0,C 180,E1 -16566.918,E2 -16566.918} C_VEL
LIN {X 0,Y 291.568,Z 548.16,A -85,B 0,C 180,E1 -16569.714,E2 -16569.714} C_VEL
LIN {X 0,Y 291.515,Z 548.161,A -85,B 0,C 180,E1 -16573.951,E2 -16573.951} C_VEL
LIN {X 0,Y 291.48,Z 548.175,A -85,B 0,C 180,E1 -16576.818,E2 -16576.818} C_VEL
LIN {X 0,Y 291.445,Z 548.178,A -85,B 0,C 180,E1 -16579.875,E2 -16579.875} C_VEL
LIN {X 0,Y 291.377,Z 548.186,A -85,B 0,C 180,E1 -16584.207,E2 -16584.207} C_VEL
LIN {X 0,Y 291.417,Z 548.176,A -85,B 0,C 180,E1 -16587.272,E2 -16587.272} C_VEL
LIN {X 0,Y 291.332,Z 548.195,A -85,B 0,C 180,E1 -16590.437,E2 -16590.437} C_VEL
LIN {X 0,Y 291.34,Z 548.193,A -85,B 0,C 180,E1 -16593.699,E2 -16593.699} C_VEL
LIN {X 0,Y 291.394,Z 548.187,A -85,B 0,C 180,E1 -16597.26,E2 -16597.26} C_VEL
LIN {X 0,Y 291.373,Z 548.192,A -85,B 0,C 180,E1 -16600.636,E2 -16600.636} C_VEL
LIN {X 0,Y 291.321,Z 548.199,A -85,B 0,C 180,E1 -16604.396,E2 -16604.396} C_VEL
LIN {X 0,Y 291.324,Z 548.198,A -85,B 0,C 180,E1 -16608.405,E2 -16608.405} C_VEL
LIN {X 0,Y 291.351,Z 548.195,A -85,B 0,C 180,E1 -16611.159,E2 -16611.159} C_VEL
LIN {X 0,Y 291.416,Z 548.383,A -85,B 0,C 180,E1 -16613.997,E2 -16613.997} C_VEL
LIN {X 0,Y 293.747,Z 558.163,A -85,B 0,C 180,E1 -16617.641,E2 -16617.641} C_VEL
LIN {X 0,Y 295.924,Z 568.01,A -85,B 0,C 180,E1 -16621.089,E2 -16621.089} C_VEL
LIN {X 0,Y 296.076,Z 568.779,A -85,B 0,C 180,E1 -16621.309,E2 -16621.309} C_VEL
LIN {X 0,Y 301.137,Z 580.952,A -85,B 0,C 180,E1 -16622.196,E2 -16622.196} C_VEL
LIN {X 0,Y 306.145,Z 608.492,A -85,B 0,C 180,E1 -16623.442,E2 -16623.442} C_VEL
LIN {X 0,Y 306.781,Z 614.248,A -85,B 0,C 180,E1 -16623.655,E2 -16623.655} C_VEL
LIN {X 0,Y 304.939,Z 677,A -85,B 0,C 180,E1 -16625.136,E2 -16625.136} C_VEL
LIN {X 0,Y 303.988,Z 690.054,A -85,B 0,C 180,E1 -16625.682,E2 -16625.682} C_VEL
LIN {X 0,Y 302.596,Z 702.776,A -85,B 0,C 180,E1 -16626.473,E2 -16626.473} C_VEL
LIN {X 0,Y 301.052,Z 714.877,A -85,B 0,C 180,E1 -16627.526,E2 -16627.526} C_VEL
LIN {X 0,Y 299.142,Z 726.388,A -85,B 0,C 180,E1 -16628.826,E2 -16628.826} C_VEL
LIN {X 0,Y 297.277,Z 736.765,A -85,B 0,C 180,E1 -16630.313,E2 -16630.313} C_VEL
LIN {X 0,Y 295.474,Z 746.11,A -85,B 0,C 180,E1 -16631.989,E2 -16631.989} C_VEL
LIN {X 0,Y 293.755,Z 755.153,A -85,B 0,C 180,E1 -16634.03,E2 -16634.03} C_VEL
LIN {X 0,Y 292.223,Z 762.453,A -85,B 0,C 180,E1 -16636.084,E2 -16636.084} C_VEL
LIN {X 0,Y 291.086,Z 768.315,A -85,B 0,C 180,E1 -16638.158,E2 -16638.158} C_VEL
LIN {X 0,Y 290.284,Z 772.945,A -85,B 0,C 180,E1 -16640.243,E2 -16640.243} C_VEL
LIN {X 0,Y 289.739,Z 776.478,A -85,B 0,C 180,E1 -16642.334,E2 -16642.334} C_VEL
LIN {X 0,Y 289.475,Z 779.105,A -85,B 0,C 180,E1 -16644.513,E2 -16644.513} C_VEL
LIN {X 0,Y 289.43,Z 780.206,A -85,B 0,C 180,E1 -16645.823,E2 -16645.823} C_VEL
LIN {X 0,Y 289.438,Z 780.958,A -85,B 0,C 180,E1 -16647.217,E2 -16647.217} C_VEL
LIN {X 0,Y 289.415,Z 781.319,A -85,B 0,C 180,E1 -16648.609,E2 -16648.609} C_VEL
LIN {X 0,Y 289.437,Z 781.296,A -85,B 0,C 180,E1 -16650,E2 -16650} C_VEL
LIN {X 0,Y 289.416,Z 780.882,A -85,B 0,C 180,E1 -16651.391,E2 -16651.391} C_VEL
LIN {X 0,Y 289.439,Z 780.032,A -85,B 0,C 180,E1 -16652.783,E2 -16652.783} C_VEL
LIN {X 0,Y 289.478,Z 777.21,A -85,B 0,C 180,E1 -16655.494,E2 -16655.494} C_VEL
LIN {X 0,Y 289.717,Z 773.757,A -85,B 0,C 180,E1 -16657.667,E2 -16657.667} C_VEL
LIN {X 0,Y 290.17,Z 769.325,A -85,B 0,C 180,E1 -16659.761,E2 -16659.761} C_VEL
LIN {X 0,Y 290.858,Z 763.687,A -85,B 0,C 180,E1 -16661.852,E2 -16661.852} C_VEL
LIN {X 0,Y 291.981,Z 756.64,A -85,B 0,C 180,E1 -16663.928,E2 -16663.928} C_VEL
LIN {X 0,Y 293.409,Z 747.812,A -85,B 0,C 180,E1 -16665.989,E2 -16665.989} C_VEL
LIN {X 0,Y 294.782,Z 737.986,A -85,B 0,C 180,E1 -16667.837,E2 -16667.837} C_VEL
LIN {X 0,Y 296.304,Z 727.521,A -85,B 0,C 180,E1 -16669.394,E2 -16669.394} C_VEL
LIN {X 0,Y 297.831,Z 716.144,A -85,B 0,C 180,E1 -16670.729,E2 -16670.729} C_VEL
LIN {X 0,Y 299.16,Z 704.321,A -85,B 0,C 180,E1 -16671.806,E2 -16671.806} C_VEL
LIN {X 0,Y 300.307,Z 692.089,A -85,B 0,C 180,E1 -16672.623,E2 -16672.623} C_VEL
LIN {X 0,Y 301.22,Z 678.508,A -85,B 0,C 180,E1 -16673.231,E2 -16673.231} C_VEL
LIN {X 0,Y 302.136,Z 645.839,A -85,B 0,C 180,E1 -16674.036,E2 -16674.036} C_VEL
LIN {X 0,Y 302.827,Z 610.801,A -85,B 0,C 180,E1 -16674.865,E2 -16674.865} C_VEL
LIN {X 0,Y 298.339,Z 580.436,A -85,B 0,C 180,E1 -16676.012,E2 -16676.012} C_VEL
LIN {X 0,Y 296.465,Z 571.383,A -85,B 0,C 180,E1 -16676.41,E2 -16676.41} C_VEL
LIN {X 0,Y 295.656,Z 568.817,A -85,B 0,C 180,E1 -16676.574,E2 -16676.574} C_VEL
LIN {X 0,Y 293.512,Z 557.728,A -85,B 0,C 180,E1 -16680.187,E2 -16680.187} C_VEL
LIN {X 0,Y 291.407,Z 548.189,A -85,B 0,C 180,E1 -16683.529,E2 -16683.529} C_VEL
LIN {X 0,Y 291.392,Z 548.19,A -85,B 0,C 180,E1 -16687.258,E2 -16687.258} C_VEL
LIN {X 0,Y 291.332,Z 548.194,A -85,B 0,C 180,E1 -16690.641,E2 -16690.641} C_VEL
LIN {X 0,Y 291.311,Z 548.195,A -85,B 0,C 180,E1 -16694.397,E2 -16694.397} C_VEL
LIN {X 0,Y 291.353,Z 548.191,A -85,B 0,C 180,E1 -16698.397,E2 -16698.397} C_VEL
LIN {X 0,Y 291.371,Z 548.19,A -85,B 0,C 180,E1 -16701.161,E2 -16701.161} C_VEL
LIN {X 0,Y 291.381,Z 548.187,A -85,B 0,C 180,E1 -16704.629,E2 -16704.629} C_VEL
LIN {X 0,Y 291.367,Z 548.189,A -85,B 0,C 180,E1 -16707.95,E2 -16707.95} C_VEL
LIN {X 0,Y 291.377,Z 548.189,A -85,B 0,C 180,E1 -16711.158,E2 -16711.158} C_VEL
LIN {X 0,Y 291.41,Z 548.183,A -85,B 0,C 180,E1 -16714.271,E2 -16714.271} C_VEL
LIN {X 0,Y 291.368,Z 548.188,A -85,B 0,C 180,E1 -16717.299,E2 -16717.299} C_VEL
LIN {X 0,Y 291.452,Z 548.178,A -85,B 0,C 180,E1 -16720.27,E2 -16720.27} C_VEL
LIN {X 0,Y 291.534,Z 548.167,A -85,B 0,C 180,E1 -16724.634,E2 -16724.634} C_VEL
LIN {X 0,Y 291.53,Z 548.165,A -85,B 0,C 180,E1 -16728.88,E2 -16728.88} C_VEL
LIN {X 0,Y 291.7,Z 548.15,A -85,B 0,C 180,E1 -16731.688,E2 -16731.688} C_VEL
LIN {X 0,Y 291.622,Z 548.154,A -85,B 0,C 180,E1 -16734.468,E2 -16734.468} C_VEL
LIN {X 0,Y 291.883,Z 548.124,A -85,B 0,C 180,E1 -16738.62,E2 -16738.62} C_VEL
LIN {X 0,Y 291.883,Z 548.125,A -85,B 0,C 180,E1 -16741.38,E2 -16741.38} C_VEL
LIN {X 0,Y 291.729,Z 548.145,A -85,B 0,C 180,E1 -16746.919,E2 -16746.919} C_VEL
LIN {X 0,Y 291.568,Z 548.157,A -85,B 0,C 180,E1 -16749.714,E2 -16749.714} C_VEL
LIN {X 0,Y 291.515,Z 548.171,A -85,B 0,C 180,E1 -16753.951,E2 -16753.951} C_VEL
LIN {X 0,Y 291.481,Z 548.175,A -85,B 0,C 180,E1 -16756.818,E2 -16756.818} C_VEL
LIN {X 0,Y 291.446,Z 548.173,A -85,B 0,C 180,E1 -16759.875,E2 -16759.875} C_VEL
LIN {X 0,Y 291.395,Z 548.185,A -85,B 0,C 180,E1 -16764.206,E2 -16764.206} C_VEL
LIN {X 0,Y 291.418,Z 548.183,A -85,B 0,C 180,E1 -16767.272,E2 -16767.272} C_VEL
LIN {X 0,Y 291.333,Z 548.192,A -85,B 0,C 180,E1 -16770.438,E2 -16770.438} C_VEL
LIN {X 0,Y 291.341,Z 548.194,A -85,B 0,C 180,E1 -16773.699,E2 -16773.699} C_VEL
LIN {X 0,Y 291.386,Z 548.182,A -85,B 0,C 180,E1 -16777.258,E2 -16777.258} C_VEL
LIN {X 0,Y 291.347,Z 548.191,A -85,B 0,C 180,E1 -16780.641,E2 -16780.641} C_VEL
LIN {X 0,Y 291.34,Z 548.192,A -85,B 0,C 180,E1 -16784.393,E2 -16784.393} C_VEL
LIN {X 0,Y 291.385,Z 548.185,A -85,B 0,C 180,E1 -16788.392,E2 -16788.392} C_VEL
LIN {X 0,Y 291.384,Z 548.189,A -85,B 0,C 180,E1 -16791.164,E2 -16791.164} C_VEL
LIN {X 0,Y 291.386,Z 548.187,A -85,B 0,C 180,E1 -16794.63,E2 -16794.63} C_VEL
LIN {X 0,Y 291.372,Z 548.191,A -85,B 0,C 180,E1 -16797.952,E2 -16797.952} C_VEL
LIN {X 0,Y 291.386,Z 548.191,A -85,B 0,C 180,E1 -16801.16,E2 -16801.16} C_VEL
LIN {X 0,Y 291.478,Z 548.277,A -85,B 0,C 180,E1 -16805.043,E2 -16805.043} C_VEL
LIN {X 0,Y 292.709,Z 554.209,A -85,B 0,C 180,E1 -16807.257,E2 -16807.257} C_VEL
LIN {X 0,Y 301.087,Z 575.726,A -85,B 0,C 180,E1 -16808.558,E2 -16808.558} C_VEL
LIN {X 0,Y 302.279,Z 580.45,A -85,B 0,C 180,E1 -16808.779,E2 -16808.779} C_VEL
LIN {X 0,Y 303.434,Z 587.318,A -85,B 0,C 180,E1 -16809.048,E2 -16809.048} C_VEL
LIN {X 0,Y 301.602,Z 661.539,A -85,B 0,C 180,E1 -16810.816,E2 -16810.816} C_VEL
LIN {X 0,Y 300.908,Z 674.722,A -85,B 0,C 180,E1 -16811.401,E2 -16811.401} C_VEL
LIN {X 0,Y 299.946,Z 686.671,A -85,B 0,C 180,E1 -16812.178,E2 -16812.178} C_VEL
LIN {X 0,Y 298.62,Z 698.77,A -85,B 0,C 180,E1 -16813.244,E2 -16813.244} C_VEL
LIN {X 0,Y 297.27,Z 710.228,A -85,B 0,C 180,E1 -16814.576,E2 -16814.576} C_VEL
LIN {X 0,Y 295.767,Z 720.558,A -85,B 0,C 180,E1 -16816.079,E2 -16816.079} C_VEL
LIN {X 0,Y 294.316,Z 729.014,A -85,B 0,C 180,E1 -16817.59,E2 -16817.59} C_VEL
LIN {X 0,Y 293.121,Z 737.85,A -85,B 0,C 180,E1 -16819.563,E2 -16819.563} C_VEL
LIN {X 0,Y 291.904,Z 745.506,A -85,B 0,C 180,E1 -16821.694,E2 -16821.694} C_VEL
LIN {X 0,Y 290.983,Z 751.411,A -85,B 0,C 180,E1 -16823.761,E2 -16823.761} C_VEL
LIN {X 0,Y 290.179,Z 756.085,A -85,B 0,C 180,E1 -16825.833,E2 -16825.833} C_VEL
LIN {X 0,Y 289.832,Z 759.653,A -85,B 0,C 180,E1 -16827.916,E2 -16827.916} C_VEL
LIN {X 0,Y 289.498,Z 762.23,A -85,B 0,C 180,E1 -16830,E2 -16830} C_VEL
LIN {X 0,Y 289.453,Z 763.443,A -85,B 0,C 180,E1 -16831.391,E2 -16831.391} C_VEL
LIN {X 0,Y 289.483,Z 764.236,A -85,B 0,C 180,E1 -16832.783,E2 -16832.783} C_VEL
LIN {X 0,Y 289.482,Z 764.631,A -85,B 0,C 180,E1 -16835.573,E2 -16835.573} C_VEL
LIN {X 0,Y 289.547,Z 764.259,A -85,B 0,C 180,E1 -16836.971,E2 -16836.971} C_VEL
LIN {X 0,Y 289.643,Z 763.479,A -85,B 0,C 180,E1 -16838.371,E2 -16838.371} C_VEL
LIN {X 0,Y 289.838,Z 762.27,A -85,B 0,C 180,E1 -16839.772,E2 -16839.772} C_VEL
LIN {X 0,Y 290.33,Z 759.695,A -85,B 0,C 180,E1 -16841.874,E2 -16841.874} C_VEL
LIN {X 0,Y 291.02,Z 756.106,A -85,B 0,C 180,E1 -16843.974,E2 -16843.974} C_VEL
LIN {X 0,Y 292.019,Z 751.395,A -85,B 0,C 180,E1 -16846.066,E2 -16846.066} C_VEL
LIN {X 0,Y 293.288,Z 745.414,A -85,B 0,C 180,E1 -16848.15,E2 -16848.15} C_VEL
LIN {X 0,Y 294.886,Z 737.95,A -85,B 0,C 180,E1 -16850.217,E2 -16850.217} C_VEL
LIN {X 0,Y 296.484,Z 730.316,A -85,B 0,C 180,E1 -16851.922,E2 -16851.922} C_VEL
LIN {X 0,Y 298.177,Z 721.023,A -85,B 0,C 180,E1 -16853.621,E2 -16853.621} C_VEL
LIN {X 0,Y 300.006,Z 710.644,A -85,B 0,C 180,E1 -16855.125,E2 -16855.125} C_VEL
LIN {X 0,Y 301.793,Z 699.101,A -85,B 0,C 180,E1 -16856.447,E2 -16856.447} C_VEL
LIN {X 0,Y 303.289,Z 686.935,A -85,B 0,C 180,E1 -16857.516,E2 -16857.516} C_VEL
LIN {X 0,Y 304.393,Z 675.035,A -85,B 0,C 180,E1 -16858.284,E2 -16858.284} C_VEL
LIN {X 0,Y 305.255,Z 662.114,A -85,B 0,C 180,E1 -16858.85,E2 -16858.85} C_VEL
LIN {X 0,Y 306.818,Z 610.51,A -85,B 0,C 180,E1 -16860.084,E2 -16860.084} C_VEL
LIN {X 0,Y 307.369,Z 588.994,A -85,B 0,C 180,E1 -16860.588,E2 -16860.588} C_VEL
LIN {X 0,Y 306,Z 583.923,A -85,B 0,C 180,E1 -16860.86,E2 -16860.86} C_VEL
LIN {X 0,Y 299.227,Z 568.055,A -85,B 0,C 180,E1 -16862.004,E2 -16862.004} C_VEL
LIN {X 0,Y 292.843,Z 554.427,A -85,B 0,C 180,E1 -16863.131,E2 -16863.131} C_VEL
LIN {X 0,Y 291.377,Z 548.189,A -85,B 0,C 180,E1 -16865.689,E2 -16865.689} C_VEL
LIN {X 0,Y 291.403,Z 548.188,A -85,B 0,C 180,E1 -16869.486,E2 -16869.486} C_VEL
LIN {X 0,Y 291.369,Z 548.189,A -85,B 0,C 180,E1 -16873.645,E2 -16873.645} C_VEL
LIN {X 0,Y 291.352,Z 548.189,A -85,B 0,C 180,E1 -16877.513,E2 -16877.513} C_VEL
LIN {X 0,Y 291.378,Z 548.191,A -85,B 0,C 180,E1 -16881.162,E2 -16881.162} C_VEL
LIN {X 0,Y 291.383,Z 548.192,A -85,B 0,C 180,E1 -16884.629,E2 -16884.629} C_VEL
LIN {X 0,Y 291.362,Z 548.191,A -85,B 0,C 180,E1 -16887.888,E2 -16887.888} C_VEL
LIN {X 0,Y 290.78,Z 548.266,A -85,B 0,C 180,E1 -16889.042,E2 -16889.042} C_VEL
LIN {X 0,Y 287.972,Z 548.615,A -85,B 0,C 180,E1 -16890.922,E2 -16890.922} C_VEL
LIN {X 0,Y 285.523,Z 548.917,A -85,B 0,C 180,E1 -16892.447,E2 -16892.447} C_VEL
LIN {X 0,Y 284.443,Z 549.045,A -85,B 0,C 180,E1 -16893.629,E2 -16893.629} C_VEL
LIN {X 0,Y 284.343,Z 549.057,A -85,B 0,C 180,E1 -16894.03,E2 -16894.03} C_VEL
LIN {X 0,Y 284.361,Z 549.059,A -85,B 0,C 180,E1 -16896.706,E2 -16896.706} C_VEL
LIN {X 0,Y 284.397,Z 549.054,A -85,B 0,C 180,E1 -16901.261,E2 -16901.261} C_VEL
LIN {X 0,Y 284.487,Z 549.048,A -85,B 0,C 180,E1 -16904.459,E2 -16904.459} C_VEL
LIN {X 0,Y 284.481,Z 549.044,A -85,B 0,C 180,E1 -16908.601,E2 -16908.601} C_VEL
LIN {X 0,Y 284.633,Z 549.023,A -85,B 0,C 180,E1 -16911.48,E2 -16911.48} C_VEL
LIN {X 0,Y 284.592,Z 549.032,A -85,B 0,C 180,E1 -16914.331,E2 -16914.331} C_VEL
LIN {X 0,Y 284.85,Z 548.993,A -85,B 0,C 180,E1 -16918.586,E2 -16918.586} C_VEL
LIN {X 0,Y 284.85,Z 549,A -85,B 0,C 180,E1 -16921.414,E2 -16921.414} C_VEL
LIN {X 0,Y 284.68,Z 549.019,A -85,B 0,C 180,E1 -16927.09,E2 -16927.09} C_VEL
LIN {X 0,Y 284.513,Z 549.04,A -85,B 0,C 180,E1 -16929.957,E2 -16929.957} C_VEL
LIN {X 0,Y 284.471,Z 549.04,A -85,B 0,C 180,E1 -16934.303,E2 -16934.303} C_VEL
LIN {X 0,Y 284.419,Z 549.052,A -85,B 0,C 180,E1 -16937.249,E2 -16937.249} C_VEL
LIN {X 0,Y 284.372,Z 549.061,A -85,B 0,C 180,E1 -16940.243,E2 -16940.243} C_VEL
LIN {X 0,Y 284.333,Z 549.068,A -85,B 0,C 180,E1 -16944.847,E2 -16944.847} C_VEL
LIN {X 0,Y 284.327,Z 549.061,A -85,B 0,C 180,E1 -16948.011,E2 -16948.011} C_VEL
LIN {X 0,Y 284.291,Z 549.071,A -85,B 0,C 180,E1 -16951.275,E2 -16951.275} C_VEL
LIN {X 0,Y 284.357,Z 549.063,A -85,B 0,C 180,E1 -16955.354,E2 -16955.354} C_VEL
LIN {X 0,Y 284.325,Z 549.068,A -85,B 0,C 180,E1 -16958.167,E2 -16958.167} C_VEL
LIN {X 0,Y 284.299,Z 549.073,A -85,B 0,C 180,E1 -16961.871,E2 -16961.871} C_VEL
LIN {X 0,Y 284.263,Z 549.076,A -85,B 0,C 180,E1 -16965.806,E2 -16965.806} C_VEL
LIN {X 0,Y 284.304,Z 549.072,A -85,B 0,C 180,E1 -16970.025,E2 -16970.025} C_VEL
LIN {X 0,Y 284.377,Z 549.263,A -85,B 0,C 180,E1 -16973.291,E2 -16973.291} C_VEL
LIN {X 0,Y 286.589,Z 558.456,A -85,B 0,C 180,E1 -16976.844,E2 -16976.844} C_VEL
LIN {X 0,Y 288.693,Z 567.733,A -85,B 0,C 180,E1 -16980.222,E2 -16980.222} C_VEL
LIN {X 0,Y 288.882,Z 568.675,A -85,B 0,C 180,E1 -16980.47,E2 -16980.47} C_VEL
LIN {X 0,Y 295.218,Z 583.689,A -85,B 0,C 180,E1 -16981.623,E2 -16981.623} C_VEL
LIN {X 0,Y 299.475,Z 607.049,A -85,B 0,C 180,E1 -16982.719,E2 -16982.719} C_VEL
LIN {X 0,Y 300.512,Z 614.678,A -85,B 0,C 180,E1 -16983.032,E2 -16983.032} C_VEL
LIN {X 0,Y 298.594,Z 676.941,A -85,B 0,C 180,E1 -16984.531,E2 -16984.531} C_VEL
LIN {X 0,Y 297.56,Z 690.594,A -85,B 0,C 180,E1 -16985.121,E2 -16985.121} C_VEL
LIN {X 0,Y 296.124,Z 703.119,A -85,B 0,C 180,E1 -16985.927,E2 -16985.927} C_VEL
LIN {X 0,Y 294.513,Z 715.057,A -85,B 0,C 180,E1 -16986.999,E2 -16986.999} C_VEL
LIN {X 0,Y 292.547,Z 726.498,A -85,B 0,C 180,E1 -16988.324,E2 -16988.324} C_VEL
LIN {X 0,Y 290.61,Z 736.82,A -85,B 0,C 180,E1 -16989.842,E2 -16989.842} C_VEL
LIN {X 0,Y 288.717,Z 746.103,A -85,B 0,C 180,E1 -16991.552,E2 -16991.552} C_VEL
LIN {X 0,Y 286.885,Z 755.112,A -85,B 0,C 180,E1 -16993.637,E2 -16993.637} C_VEL
LIN {X 0,Y 285.317,Z 762.383,A -85,B 0,C 180,E1 -16995.74,E2 -16995.74} C_VEL
LIN {X 0,Y 284.106,Z 768.218,A -85,B 0,C 180,E1 -16997.862,E2 -16997.862} C_VEL
LIN {X 0,Y 283.249,Z 772.824,A -85,B 0,C 180,E1 -16999.998,E2 -16999.998} C_VEL
LIN {X 0,Y 282.696,Z 776.337,A -85,B 0,C 180,E1 -17002.141,E2 -17002.141} C_VEL
LIN {X 0,Y 282.369,Z 779.159,A -85,B 0,C 180,E1 -17004.609,E2 -17004.609} C_VEL
LIN {X 0,Y 282.345,Z 780.767,A -85,B 0,C 180,E1 -17007.147,E2 -17007.147} C_VEL
LIN {X 0,Y 282.338,Z 781.12,A -85,B 0,C 180,E1 -17008.574,E2 -17008.574} C_VEL
LIN {X 0,Y 282.357,Z 781.087,A -85,B 0,C 180,E1 -17010,E2 -17010} C_VEL
LIN {X 0,Y 282.339,Z 780.659,A -85,B 0,C 180,E1 -17011.426,E2 -17011.426} C_VEL
LIN {X 0,Y 282.346,Z 779.793,A -85,B 0,C 180,E1 -17012.853,E2 -17012.853} C_VEL
LIN {X 0,Y 282.402,Z 777.169,A -85,B 0,C 180,E1 -17015.46,E2 -17015.46} C_VEL
LIN {X 0,Y 282.673,Z 773.477,A -85,B 0,C 180,E1 -17017.859,E2 -17017.859} C_VEL
LIN {X 0,Y 283.148,Z 769.022,A -85,B 0,C 180,E1 -17020.005,E2 -17020.005} C_VEL
LIN {X 0,Y 283.873,Z 763.359,A -85,B 0,C 180,E1 -17022.148,E2 -17022.148} C_VEL
LIN {X 0,Y 285.079,Z 756.272,A -85,B 0,C 180,E1 -17024.272,E2 -17024.272} C_VEL
LIN {X 0,Y 286.571,Z 747.409,A -85,B 0,C 180,E1 -17026.381,E2 -17026.381} C_VEL
LIN {X 0,Y 288.016,Z 737.369,A -85,B 0,C 180,E1 -17028.301,E2 -17028.301} C_VEL
LIN {X 0,Y 289.583,Z 726.999,A -85,B 0,C 180,E1 -17029.862,E2 -17029.862} C_VEL
LIN {X 0,Y 291.168,Z 715.55,A -85,B 0,C 180,E1 -17031.226,E2 -17031.226} C_VEL
LIN {X 0,Y 292.534,Z 703.615,A -85,B 0,C 180,E1 -17032.326,E2 -17032.326} C_VEL
LIN {X 0,Y 293.766,Z 691.141,A -85,B 0,C 180,E1 -17033.156,E2 -17033.156} C_VEL
LIN {X 0,Y 294.699,Z 677.19,A -85,B 0,C 180,E1 -17033.777,E2 -17033.777} C_VEL
LIN {X 0,Y 296.354,Z 612.075,A -85,B 0,C 180,E1 -17035.362,E2 -17035.362} C_VEL
LIN {X 0,Y 292.201,Z 583.549,A -85,B 0,C 180,E1 -17036.468,E2 -17036.468} C_VEL
LIN {X 0,Y 290.289,Z 573.944,A -85,B 0,C 180,E1 -17036.897,E2 -17036.897} C_VEL
LIN {X 0,Y 288.41,Z 568.567,A -85,B 0,C 180,E1 -17037.25,E2 -17037.25} C_VEL
LIN {X 0,Y 286.344,Z 558.053,A -85,B 0,C 180,E1 -17040.791,E2 -17040.791} C_VEL
LIN {X 0,Y 284.353,Z 549.067,A -85,B 0,C 180,E1 -17043.998,E2 -17043.998} C_VEL
LIN {X 0,Y 284.321,Z 549.068,A -85,B 0,C 180,E1 -17048.166,E2 -17048.166} C_VEL
LIN {X 0,Y 284.267,Z 549.074,A -85,B 0,C 180,E1 -17052.124,E2 -17052.124} C_VEL
LIN {X 0,Y 284.286,Z 549.07,A -85,B 0,C 180,E1 -17056.195,E2 -17056.195} C_VEL
LIN {X 0,Y 284.348,Z 549.064,A -85,B 0,C 180,E1 -17060.012,E2 -17060.012} C_VEL
LIN {X 0,Y 284.347,Z 549.065,A -85,B 0,C 180,E1 -17063.616,E2 -17063.616} C_VEL
LIN {X 0,Y 284.303,Z 549.069,A -85,B 0,C 180,E1 -17067.189,E2 -17067.189} C_VEL
LIN {X 0,Y 284.354,Z 549.062,A -85,B 0,C 180,E1 -17070.376,E2 -17070.376} C_VEL
LIN {X 0,Y 284.372,Z 549.064,A -85,B 0,C 180,E1 -17073.586,E2 -17073.586} C_VEL
LIN {X 0,Y 284.327,Z 549.063,A -85,B 0,C 180,E1 -17076.704,E2 -17076.704} C_VEL
LIN {X 0,Y 284.393,Z 549.06,A -85,B 0,C 180,E1 -17081.261,E2 -17081.261} C_VEL
LIN {X 0,Y 284.472,Z 549.047,A -85,B 0,C 180,E1 -17084.469,E2 -17084.469} C_VEL
LIN {X 0,Y 284.481,Z 549.041,A -85,B 0,C 180,E1 -17088.601,E2 -17088.601} C_VEL
LIN {X 0,Y 284.651,Z 549.03,A -85,B 0,C 180,E1 -17091.481,E2 -17091.481} C_VEL
LIN {X 0,Y 284.593,Z 549.029,A -85,B 0,C 180,E1 -17094.331,E2 -17094.331} C_VEL
LIN {X 0,Y 284.849,Z 549.001,A -85,B 0,C 180,E1 -17098.586,E2 -17098.586} C_VEL
LIN {X 0,Y 284.849,Z 549,A -85,B 0,C 180,E1 -17101.414,E2 -17101.414} C_VEL
LIN {X 0,Y 284.68,Z 549.024,A -85,B 0,C 180,E1 -17107.091,E2 -17107.091} C_VEL
LIN {X 0,Y 284.513,Z 549.034,A -85,B 0,C 180,E1 -17109.957,E2 -17109.957} C_VEL
LIN {X 0,Y 284.472,Z 549.047,A -85,B 0,C 180,E1 -17114.304,E2 -17114.304} C_VEL
LIN {X 0,Y 284.419,Z 549.057,A -85,B 0,C 180,E1 -17117.249,E2 -17117.249} C_VEL
LIN {X 0,Y 284.375,Z 549.051,A -85,B 0,C 180,E1 -17120.243,E2 -17120.243} C_VEL
LIN {X 0,Y 284.364,Z 549.063,A -85,B 0,C 180,E1 -17123.876,E2 -17123.876} C_VEL
LIN {X 0,Y 284.393,Z 549.057,A -85,B 0,C 180,E1 -17127.174,E2 -17127.174} C_VEL
LIN {X 0,Y 284.292,Z 549.072,A -85,B 0,C 180,E1 -17131.275,E2 -17131.275} C_VEL
LIN {X 0,Y 284.358,Z 549.063,A -85,B 0,C 180,E1 -17135.355,E2 -17135.355} C_VEL
LIN {X 0,Y 284.313,Z 549.061,A -85,B 0,C 180,E1 -17138.169,E2 -17138.169} C_VEL
LIN {X 0,Y 284.294,Z 549.069,A -85,B 0,C 180,E1 -17142.131,E2 -17142.131} C_VEL
LIN {X 0,Y 284.316,Z 549.066,A -85,B 0,C 180,E1 -17146.202,E2 -17146.202} C_VEL
LIN {X 0,Y 284.35,Z 549.063,A -85,B 0,C 180,E1 -17150.014,E2 -17150.014} C_VEL
LIN {X 0,Y 284.355,Z 549.064,A -85,B 0,C 180,E1 -17153.618,E2 -17153.618} C_VEL
LIN {X 0,Y 284.308,Z 549.072,A -85,B 0,C 180,E1 -17157.19,E2 -17157.19} C_VEL
LIN {X 0,Y 284.36,Z 549.065,A -85,B 0,C 180,E1 -17160.377,E2 -17160.377} C_VEL
LIN {X 0,Y 284.407,Z 549.083,A -85,B 0,C 180,E1 -17164.525,E2 -17164.525} C_VEL
LIN {X 0,Y 285.503,Z 554.332,A -85,B 0,C 180,E1 -17166.548,E2 -17166.548} C_VEL
LIN {X 0,Y 294.596,Z 577.321,A -85,B 0,C 180,E1 -17168.038,E2 -17168.038} C_VEL
LIN {X 0,Y 295.884,Z 581.967,A -85,B 0,C 180,E1 -17168.272,E2 -17168.272} C_VEL
LIN {X 0,Y 296.925,Z 588.344,A -85,B 0,C 180,E1 -17168.528,E2 -17168.528} C_VEL
LIN {X 0,Y 295.042,Z 661.278,A -85,B 0,C 180,E1 -17170.295,E2 -17170.295} C_VEL
LIN {X 0,Y 294.348,Z 674.399,A -85,B 0,C 180,E1 -17170.88,E2 -17170.88} C_VEL
LIN {X 0,Y 293.35,Z 686.483,A -85,B 0,C 180,E1 -17171.673,E2 -17171.673} C_VEL
LIN {X 0,Y 292.086,Z 697.888,A -85,B 0,C 180,E1 -17172.677,E2 -17172.677} C_VEL
LIN {X 0,Y 290.657,Z 709.567,A -85,B 0,C 180,E1 -17174.036,E2 -17174.036} C_VEL
LIN {X 0,Y 289.075,Z 720.046,A -85,B 0,C 180,E1 -17175.57,E2 -17175.57} C_VEL
LIN {X 0,Y 287.404,Z 729.505,A -85,B 0,C 180,E1 -17177.287,E2 -17177.287} C_VEL
LIN {X 0,Y 286.116,Z 738.673,A -85,B 0,C 180,E1 -17179.41,E2 -17179.41} C_VEL
LIN {X 0,Y 284.898,Z 745.892,A -85,B 0,C 180,E1 -17181.489,E2 -17181.489} C_VEL
LIN {X 0,Y 283.949,Z 751.762,A -85,B 0,C 180,E1 -17183.605,E2 -17183.605} C_VEL
LIN {X 0,Y 283.119,Z 756.405,A -85,B 0,C 180,E1 -17185.729,E2 -17185.729} C_VEL
LIN {X 0,Y 282.742,Z 759.945,A -85,B 0,C 180,E1 -17187.863,E2 -17187.863} C_VEL
LIN {X 0,Y 282.415,Z 762.493,A -85,B 0,C 180,E1 -17190,E2 -17190} C_VEL
LIN {X 0,Y 282.374,Z 763.692,A -85,B 0,C 180,E1 -17191.426,E2 -17191.426} C_VEL
LIN {X 0,Y 282.388,Z 764.46,A -85,B 0,C 180,E1 -17192.853,E2 -17192.853} C_VEL
LIN {X 0,Y 282.378,Z 764.863,A -85,B 0,C 180,E1 -17195.405,E2 -17195.405} C_VEL
LIN {X 0,Y 282.465,Z 764.445,A -85,B 0,C 180,E1 -17197.146,E2 -17197.146} C_VEL
LIN {X 0,Y 282.576,Z 763.638,A -85,B 0,C 180,E1 -17198.582,E2 -17198.582} C_VEL
LIN {X 0,Y 283.081,Z 760.793,A -85,B 0,C 180,E1 -17201.456,E2 -17201.456} C_VEL
LIN {X 0,Y 283.809,Z 757.519,A -85,B 0,C 180,E1 -17203.606,E2 -17203.606} C_VEL
LIN {X 0,Y 284.787,Z 753.165,A -85,B 0,C 180,E1 -17205.751,E2 -17205.751} C_VEL
LIN {X 0,Y 285.973,Z 747.606,A -85,B 0,C 180,E1 -17207.89,E2 -17207.89} C_VEL
LIN {X 0,Y 287.543,Z 740.642,A -85,B 0,C 180,E1 -17210.009,E2 -17210.009} C_VEL
LIN {X 0,Y 289.544,Z 731.886,A -85,B 0,C 180,E1 -17212.1,E2 -17212.1} C_VEL
LIN {X 0,Y 291.268,Z 722.776,A -85,B 0,C 180,E1 -17213.861,E2 -17213.861} C_VEL
LIN {X 0,Y 293.107,Z 712.987,A -85,B 0,C 180,E1 -17215.378,E2 -17215.378} C_VEL
LIN {X 0,Y 294.908,Z 701.966,A -85,B 0,C 180,E1 -17216.731,E2 -17216.731} C_VEL
LIN {X 0,Y 296.63,Z 689.587,A -85,B 0,C 180,E1 -17217.9,E2 -17217.9} C_VEL
LIN {X 0,Y 297.747,Z 678.462,A -85,B 0,C 180,E1 -17218.697,E2 -17218.697} C_VEL
LIN {X 0,Y 298.748,Z 665.779,A -85,B 0,C 180,E1 -17219.331,E2 -17219.331} C_VEL
LIN {X 0,Y 299.434,Z 649.813,A -85,B 0,C 180,E1 -17219.789,E2 -17219.789} C_VEL
LIN {X 0,Y 301.127,Z 590.238,A -85,B 0,C 180,E1 -17221.201,E2 -17221.201} C_VEL
LIN {X 0,Y 299.571,Z 585.33,A -85,B 0,C 180,E1 -17221.499,E2 -17221.499} C_VEL
LIN {X 0,Y 291.778,Z 567.424,A -85,B 0,C 180,E1 -17222.867,E2 -17222.867} C_VEL
LIN {X 0,Y 285.649,Z 554.669,A -85,B 0,C 180,E1 -17223.998,E2 -17223.998} C_VEL
LIN {X 0,Y 284.364,Z 549.068,A -85,B 0,C 180,E1 -17226.38,E2 -17226.38} C_VEL
LIN {X 0,Y 284.35,Z 549.066,A -85,B 0,C 180,E1 -17229.986,E2 -17229.986} C_VEL
LIN {X 0,Y 284.316,Z 549.068,A -85,B 0,C 180,E1 -17233.798,E2 -17233.798} C_VEL
LIN {X 0,Y 284.3,Z 549.062,A -85,B 0,C 180,E1 -17237.867,E2 -17237.867} C_VEL
LIN {X 0,Y 284.349,Z 549.055,A -85,B 0,C 180,E1 -17240.012,E2 -17240.012} C_VEL
LIN {X 0,Y 284.352,Z 549.062,A -85,B 0,C 180,E1 -17243.617,E2 -17243.617} C_VEL
LIN {X 0,Y 284.273,Z 549.07,A -85,B 0,C 180,E1 -17247.885,E2 -17247.885} C_VEL
LIN {X 0,Y 284.355,Z 549.059,A -85,B 0,C 180,E1 -17250.375,E2 -17250.375} C_VEL
LIN {X 0,Y 284.343,Z 549.057,A -85,B 0,C 180,E1 -17254.03,E2 -17254.03} C_VEL
LIN {X 0,Y 283.645,Z 549.153,A -85,B 0,C 180,E1 -17255.212,E2 -17255.212} C_VEL
LIN {X 0,Y 280.799,Z 549.504,A -85,B 0,C 180,E1 -17257.137,E2 -17257.137} C_VEL
LIN {X 0,Y 278.414,Z 549.801,A -85,B 0,C 180,E1 -17258.701,E2 -17258.701} C_VEL
LIN {X 0,Y 277.404,Z 549.93,A -85,B 0,C 180,E1 -17259.912,E2 -17259.912} C_VEL
LIN {X 0,Y 277.327,Z 549.937,A -85,B 0,C 180,E1 -17260.322,E2 -17260.322} C_VEL
LIN {X 0,Y 277.438,Z 549.925,A -85,B 0,C 180,E1 -17264.277,E2 -17264.277} C_VEL
LIN {X 0,Y 277.428,Z 549.92,A -85,B 0,C 180,E1 -17268.307,E2 -17268.307} C_VEL
LIN {X 0,Y 277.592,Z 549.901,A -85,B 0,C 180,E1 -17271.262,E2 -17271.262} C_VEL
LIN {X 0,Y 277.562,Z 549.907,A -85,B 0,C 180,E1 -17274.187,E2 -17274.187} C_VEL
LIN {X 0,Y 277.816,Z 549.869,A -85,B 0,C 180,E1 -17278.55,E2 -17278.55} C_VEL
LIN {X 0,Y 277.816,Z 549.876,A -85,B 0,C 180,E1 -17281.449,E2 -17281.449} C_VEL
LIN {X 0,Y 277.634,Z 549.896,A -85,B 0,C 180,E1 -17287.271,E2 -17287.271} C_VEL
LIN {X 0,Y 277.455,Z 549.92,A -85,B 0,C 180,E1 -17290.213,E2 -17290.213} C_VEL
LIN {X 0,Y 277.422,Z 549.922,A -85,B 0,C 180,E1 -17294.675,E2 -17294.675} C_VEL
LIN {X 0,Y 277.339,Z 549.934,A -85,B 0,C 180,E1 -17299.234,E2 -17299.234} C_VEL
LIN {X 0,Y 277.286,Z 549.94,A -85,B 0,C 180,E1 -17304.158,E2 -17304.158} C_VEL
LIN {X 0,Y 277.321,Z 549.931,A -85,B 0,C 180,E1 -17307.506,E2 -17307.506} C_VEL
LIN {X 0,Y 277.267,Z 549.947,A -85,B 0,C 180,E1 -17310.482,E2 -17310.482} C_VEL
LIN {X 0,Y 277.25,Z 549.949,A -85,B 0,C 180,E1 -17313.895,E2 -17313.895} C_VEL
LIN {X 0,Y 277.281,Z 549.945,A -85,B 0,C 180,E1 -17317.467,E2 -17317.467} C_VEL
LIN {X 0,Y 277.237,Z 549.952,A -85,B 0,C 180,E1 -17321.232,E2 -17321.232} C_VEL
LIN {X 0,Y 277.217,Z 549.955,A -85,B 0,C 180,E1 -17325.223,E2 -17325.223} C_VEL
LIN {X 0,Y 277.22,Z 549.953,A -85,B 0,C 180,E1 -17329.513,E2 -17329.513} C_VEL
LIN {X 0,Y 277.315,Z 550.024,A -85,B 0,C 180,E1 -17332.493,E2 -17332.493} C_VEL
LIN {X 0,Y 279.484,Z 558.96,A -85,B 0,C 180,E1 -17336.081,E2 -17336.081} C_VEL
LIN {X 0,Y 281.577,Z 568.109,A -85,B 0,C 180,E1 -17339.536,E2 -17339.536} C_VEL
LIN {X 0,Y 289.265,Z 585.929,A -85,B 0,C 180,E1 -17341.005,E2 -17341.005} C_VEL
LIN {X 0,Y 293.469,Z 609.5,A -85,B 0,C 180,E1 -17342.139,E2 -17342.139} C_VEL
LIN {X 0,Y 294.254,Z 616.005,A -85,B 0,C 180,E1 -17342.404,E2 -17342.404} C_VEL
LIN {X 0,Y 292.303,Z 676.877,A -85,B 0,C 180,E1 -17343.901,E2 -17343.901} C_VEL
LIN {X 0,Y 291.237,Z 690.381,A -85,B 0,C 180,E1 -17344.495,E2 -17344.495} C_VEL
LIN {X 0,Y 289.797,Z 702.35,A -85,B 0,C 180,E1 -17345.271,E2 -17345.271} C_VEL
LIN {X 0,Y 288.266,Z 713.658,A -85,B 0,C 180,E1 -17346.28,E2 -17346.28} C_VEL
LIN {X 0,Y 286.2,Z 725.322,A -85,B 0,C 180,E1 -17347.628,E2 -17347.628} C_VEL
LIN {X 0,Y 284.135,Z 735.81,A -85,B 0,C 180,E1 -17349.173,E2 -17349.173} C_VEL
LIN {X 0,Y 282.347,Z 744.391,A -85,B 0,C 180,E1 -17350.743,E2 -17350.743} C_VEL
LIN {X 0,Y 280.682,Z 752.313,A -85,B 0,C 180,E1 -17352.515,E2 -17352.515} C_VEL
LIN {X 0,Y 278.959,Z 760.077,A -85,B 0,C 180,E1 -17354.661,E2 -17354.661} C_VEL
LIN {X 0,Y 277.467,Z 766.307,A -85,B 0,C 180,E1 -17356.823,E2 -17356.823} C_VEL
LIN {X 0,Y 276.51,Z 771.276,A -85,B 0,C 180,E1 -17359.011,E2 -17359.011} C_VEL
LIN {X 0,Y 275.826,Z 775.124,A -85,B 0,C 180,E1 -17361.206,E2 -17361.206} C_VEL
LIN {X 0,Y 275.509,Z 777.113,A -85,B 0,C 180,E1 -17362.672,E2 -17362.672} C_VEL
LIN {X 0,Y 275.263,Z 779.179,A -85,B 0,C 180,E1 -17364.715,E2 -17364.715} C_VEL
LIN {X 0,Y 275.255,Z 780.577,A -85,B 0,C 180,E1 -17367.073,E2 -17367.073} C_VEL
LIN {X 0,Y 275.262,Z 780.921,A -85,B 0,C 180,E1 -17368.537,E2 -17368.537} C_VEL
LIN {X 0,Y 275.279,Z 780.878,A -85,B 0,C 180,E1 -17370,E2 -17370} C_VEL
LIN {X 0,Y 275.263,Z 780.434,A -85,B 0,C 180,E1 -17371.463,E2 -17371.463} C_VEL
LIN {X 0,Y 275.256,Z 779.554,A -85,B 0,C 180,E1 -17372.927,E2 -17372.927} C_VEL
LIN {X 0,Y 275.32,Z 777.139,A -85,B 0,C 180,E1 -17375.413,E2 -17375.413} C_VEL
LIN {X 0,Y 275.601,Z 773.195,A -85,B 0,C 180,E1 -17378.062,E2 -17378.062} C_VEL
LIN {X 0,Y 276.14,Z 768.718,A -85,B 0,C 180,E1 -17380.262,E2 -17380.262} C_VEL
LIN {X 0,Y 277.065,Z 761.928,A -85,B 0,C 180,E1 -17382.823,E2 -17382.823} C_VEL
LIN {X 0,Y 278.436,Z 754.538,A -85,B 0,C 180,E1 -17384.994,E2 -17384.994} C_VEL
LIN {X 0,Y 279.999,Z 745.352,A -85,B 0,C 180,E1 -17387.153,E2 -17387.153} C_VEL
LIN {X 0,Y 281.4,Z 735.781,A -85,B 0,C 180,E1 -17388.945,E2 -17388.945} C_VEL
LIN {X 0,Y 283.082,Z 725.177,A -85,B 0,C 180,E1 -17390.528,E2 -17390.528} C_VEL
LIN {X 0,Y 284.775,Z 713.331,A -85,B 0,C 180,E1 -17391.917,E2 -17391.917} C_VEL
LIN {X 0,Y 286.231,Z 700.608,A -85,B 0,C 180,E1 -17393.036,E2 -17393.036} C_VEL
LIN {X 0,Y 287.444,Z 687.891,A -85,B 0,C 180,E1 -17393.84,E2 -17393.84} C_VEL
LIN {X 0,Y 288.196,Z 675.772,A -85,B 0,C 180,E1 -17394.347,E2 -17394.347} C_VEL
LIN {X 0,Y 289.847,Z 613.7,A -85,B 0,C 180,E1 -17395.877,E2 -17395.877} C_VEL
LIN {X 0,Y 286.673,Z 590.652,A -85,B 0,C 180,E1 -17396.781,E2 -17396.781} C_VEL
LIN {X 0,Y 284.305,Z 576.837,A -85,B 0,C 180,E1 -17397.38,E2 -17397.38} C_VEL
LIN {X 0,Y 281.201,Z 568.385,A -85,B 0,C 180,E1 -17397.942,E2 -17397.942} C_VEL
LIN {X 0,Y 279.313,Z 559.061,A -85,B 0,C 180,E1 -17401.185,E2 -17401.185} C_VEL
LIN {X 0,Y 277.302,Z 549.945,A -85,B 0,C 180,E1 -17404.546,E2 -17404.546} C_VEL
LIN {X 0,Y 277.273,Z 549.946,A -85,B 0,C 180,E1 -17408.21,E2 -17408.21} C_VEL
LIN {X 0,Y 277.215,Z 549.952,A -85,B 0,C 180,E1 -17412.675,E2 -17412.675} C_VEL
LIN {X 0,Y 277.233,Z 549.949,A -85,B 0,C 180,E1 -17416.806,E2 -17416.806} C_VEL
LIN {X 0,Y 277.262,Z 549.945,A -85,B 0,C 180,E1 -17420.677,E2 -17420.677} C_VEL
LIN {X 0,Y 277.3,Z 549.941,A -85,B 0,C 180,E1 -17424.344,E2 -17424.344} C_VEL
LIN {X 0,Y 277.24,Z 549.949,A -85,B 0,C 180,E1 -17427.836,E2 -17427.836} C_VEL
LIN {X 0,Y 277.284,Z 549.944,A -85,B 0,C 180,E1 -17431.212,E2 -17431.212} C_VEL
LIN {X 0,Y 277.304,Z 549.94,A -85,B 0,C 180,E1 -17434.479,E2 -17434.479} C_VEL
LIN {X 0,Y 277.262,Z 549.947,A -85,B 0,C 180,E1 -17437.653,E2 -17437.653} C_VEL
LIN {X 0,Y 277.337,Z 549.937,A -85,B 0,C 180,E1 -17440.766,E2 -17440.766} C_VEL
LIN {X 0,Y 277.422,Z 549.929,A -85,B 0,C 180,E1 -17445.325,E2 -17445.325} C_VEL
LIN {X 0,Y 277.5,Z 549.917,A -85,B 0,C 180,E1 -17449.789,E2 -17449.789} C_VEL
LIN {X 0,Y 277.643,Z 549.899,A -85,B 0,C 180,E1 -17452.729,E2 -17452.729} C_VEL
LIN {X 0,Y 277.815,Z 549.877,A -85,B 0,C 180,E1 -17458.551,E2 -17458.551} C_VEL
LIN {X 0,Y 277.815,Z 549.875,A -85,B 0,C 180,E1 -17461.45,E2 -17461.45} C_VEL
LIN {X 0,Y 277.635,Z 549.903,A -85,B 0,C 180,E1 -17467.272,E2 -17467.272} C_VEL
LIN {X 0,Y 277.455,Z 549.911,A -85,B 0,C 180,E1 -17470.213,E2 -17470.213} C_VEL
LIN {X 0,Y 277.422,Z 549.925,A -85,B 0,C 180,E1 -17474.675,E2 -17474.675} C_VEL
LIN {X 0,Y 277.34,Z 549.93,A -85,B 0,C 180,E1 -17479.234,E2 -17479.234} C_VEL
LIN {X 0,Y 277.324,Z 549.939,A -85,B 0,C 180,E1 -17483.921,E2 -17483.921} C_VEL
LIN {X 0,Y 277.322,Z 549.94,A -85,B 0,C 180,E1 -17487.506,E2 -17487.506} C_VEL
LIN {X 0,Y 277.268,Z 549.944,A -85,B 0,C 180,E1 -17490.482,E2 -17490.482} C_VEL
LIN {X 0,Y 277.251,Z 549.948,A -85,B 0,C 180,E1 -17493.896,E2 -17493.896} C_VEL
LIN {X 0,Y 277.274,Z 549.937,A -85,B 0,C 180,E1 -17497.469,E2 -17497.469} C_VEL
LIN {X 0,Y 277.223,Z 549.954,A -85,B 0,C 180,E1 -17501.235,E2 -17501.235} C_VEL
LIN {X 0,Y 277.245,Z 549.952,A -85,B 0,C 180,E1 -17505.218,E2 -17505.218} C_VEL
LIN {X 0,Y 277.294,Z 549.944,A -85,B 0,C 180,E1 -17509.496,E2 -17509.496} C_VEL
LIN {X 0,Y 277.29,Z 549.942,A -85,B 0,C 180,E1 -17512.535,E2 -17512.535} C_VEL
LIN {X 0,Y 277.255,Z 549.948,A -85,B 0,C 180,E1 -17516.106,E2 -17516.106} C_VEL
LIN {X 0,Y 277.262,Z 549.95,A -85,B 0,C 180,E1 -17519.539,E2 -17519.539} C_VEL
LIN {X 0,Y 277.356,Z 549.935,A -85,B 0,C 180,E1 -17523.981,E2 -17523.981} C_VEL
LIN {X 0,Y 278.341,Z 554.576,A -85,B 0,C 180,E1 -17525.843,E2 -17525.843} C_VEL
LIN {X 0,Y 287.438,Z 577.062,A -85,B 0,C 180,E1 -17527.38,E2 -17527.38} C_VEL
LIN {X 0,Y 289.512,Z 583.496,A -85,B 0,C 180,E1 -17527.745,E2 -17527.745} C_VEL
LIN {X 0,Y 290.438,Z 589.178,A -85,B 0,C 180,E1 -17527.98,E2 -17527.98} C_VEL
LIN {X 0,Y 288.475,Z 661.901,A -85,B 0,C 180,E1 -17529.784,E2 -17529.784} C_VEL
LIN {X 0,Y 287.752,Z 674.824,A -85,B 0,C 180,E1 -17530.378,E2 -17530.378} C_VEL
LIN {X 0,Y 286.77,Z 686.29,A -85,B 0,C 180,E1 -17531.144,E2 -17531.144} C_VEL
LIN {X 0,Y 285.364,Z 698.623,A -85,B 0,C 180,E1 -17532.256,E2 -17532.256} C_VEL
LIN {X 0,Y 283.875,Z 710.187,A -85,B 0,C 180,E1 -17533.644,E2 -17533.644} C_VEL
LIN {X 0,Y 282.249,Z 720.595,A -85,B 0,C 180,E1 -17535.213,E2 -17535.213} C_VEL
LIN {X 0,Y 280.516,Z 729.986,A -85,B 0,C 180,E1 -17536.969,E2 -17536.969} C_VEL
LIN {X 0,Y 279.284,Z 738.325,A -85,B 0,C 180,E1 -17538.937,E2 -17538.937} C_VEL
LIN {X 0,Y 277.9,Z 746.277,A -85,B 0,C 180,E1 -17541.273,E2 -17541.273} C_VEL
LIN {X 0,Y 276.92,Z 752.113,A -85,B 0,C 180,E1 -17543.442,E2 -17543.442} C_VEL
LIN {X 0,Y 276.063,Z 756.725,A -85,B 0,C 180,E1 -17545.62,E2 -17545.62} C_VEL
LIN {X 0,Y 275.692,Z 759.182,A -85,B 0,C 180,E1 -17547.078,E2 -17547.078} C_VEL
LIN {X 0,Y 275.472,Z 761.174,A -85,B 0,C 180,E1 -17548.538,E2 -17548.538} C_VEL
LIN {X 0,Y 275.334,Z 762.756,A -85,B 0,C 180,E1 -17550,E2 -17550} C_VEL
LIN {X 0,Y 275.298,Z 763.938,A -85,B 0,C 180,E1 -17551.463,E2 -17551.463} C_VEL
LIN {X 0,Y 275.295,Z 764.684,A -85,B 0,C 180,E1 -17552.927,E2 -17552.927} C_VEL
LIN {X 0,Y 275.294,Z 765.081,A -85,B 0,C 180,E1 -17555.351,E2 -17555.351} C_VEL
LIN {X 0,Y 275.375,Z 764.629,A -85,B 0,C 180,E1 -17557.331,E2 -17557.331} C_VEL
LIN {X 0,Y 275.525,Z 763.797,A -85,B 0,C 180,E1 -17558.803,E2 -17558.803} C_VEL
LIN {X 0,Y 276.07,Z 760.926,A -85,B 0,C 180,E1 -17561.751,E2 -17561.751} C_VEL
LIN {X 0,Y 276.856,Z 757.623,A -85,B 0,C 180,E1 -17563.955,E2 -17563.955} C_VEL
LIN {X 0,Y 277.875,Z 753.24,A -85,B 0,C 180,E1 -17566.153,E2 -17566.153} C_VEL
LIN {X 0,Y 279.157,Z 747.648,A -85,B 0,C 180,E1 -17568.342,E2 -17568.342} C_VEL
LIN {X 0,Y 280.814,Z 740.631,A -85,B 0,C 180,E1 -17570.51,E2 -17570.51} C_VEL
LIN {X 0,Y 282.886,Z 731.827,A -85,B 0,C 180,E1 -17572.648,E2 -17572.648} C_VEL
LIN {X 0,Y 284.697,Z 722.787,A -85,B 0,C 180,E1 -17574.423,E2 -17574.423} C_VEL
LIN {X 0,Y 286.658,Z 712.798,A -85,B 0,C 180,E1 -17575.991,E2 -17575.991} C_VEL
LIN {X 0,Y 288.567,Z 701.659,A -85,B 0,C 180,E1 -17577.367,E2 -17577.367} C_VEL
LIN {X 0,Y 290.328,Z 689.146,A -85,B 0,C 180,E1 -17578.56,E2 -17578.56} C_VEL
LIN {X 0,Y 291.557,Z 677.228,A -85,B 0,C 180,E1 -17579.407,E2 -17579.407} C_VEL
LIN {X 0,Y 292.567,Z 663.695,A -85,B 0,C 180,E1 -17580.048,E2 -17580.048} C_VEL
LIN {X 0,Y 293.433,Z 641.625,A -85,B 0,C 180,E1 -17580.629,E2 -17580.629} C_VEL
LIN {X 0,Y 294.896,Z 591.296,A -85,B 0,C 180,E1 -17581.849,E2 -17581.849} C_VEL
LIN {X 0,Y 289.727,Z 578.591,A -85,B 0,C 180,E1 -17582.793,E2 -17582.793} C_VEL
LIN {X 0,Y 282.038,Z 562.167,A -85,B 0,C 180,E1 -17584.209,E2 -17584.209} C_VEL
LIN {X 0,Y 278.467,Z 554.931,A -85,B 0,C 180,E1 -17584.911,E2 -17584.911} C_VEL
LIN {X 0,Y 277.287,Z 549.943,A -85,B 0,C 180,E1 -17587.149,E2 -17587.149} C_VEL
LIN {X 0,Y 277.263,Z 549.948,A -85,B 0,C 180,E1 -17591.226,E2 -17591.226} C_VEL
LIN {X 0,Y 277.248,Z 549.948,A -85,B 0,C 180,E1 -17595.215,E2 -17595.215} C_VEL
LIN {X 0,Y 277.26,Z 549.933,A -85,B 0,C 180,E1 -17599.502,E2 -17599.502} C_VEL
LIN {X 0,Y 277.286,Z 549.943,A -85,B 0,C 180,E1 -17602.533,E2 -17602.533} C_VEL
LIN {X 0,Y 277.251,Z 549.945,A -85,B 0,C 180,E1 -17606.104,E2 -17606.104} C_VEL
LIN {X 0,Y 277.258,Z 549.941,A -85,B 0,C 180,E1 -17609.538,E2 -17609.538} C_VEL
LIN {X 0,Y 277.355,Z 549.93,A -85,B 0,C 180,E1 -17612.863,E2 -17612.863} C_VEL
LIN {X 0,Y 277.324,Z 549.94,A -85,B 0,C 180,E1 -17616.079,E2 -17616.079} C_VEL
LIN {X 0,Y 277.327,Z 549.937,A -85,B 0,C 180,E1 -17620.322,E2 -17620.322} C_VEL
LIN {X 0,Y 276.681,Z 550.018,A -85,B 0,C 180,E1 -17621.535,E2 -17621.535} C_VEL
LIN {X 0,Y 273.864,Z 550.371,A -85,B 0,C 180,E1 -17623.513,E2 -17623.513} C_VEL
LIN {X 0,Y 271.463,Z 550.669,A -85,B 0,C 180,E1 -17625.12,E2 -17625.12} C_VEL
LIN {X 0,Y 270.43,Z 550.793,A -85,B 0,C 180,E1 -17626.365,E2 -17626.365} C_VEL
LIN {X 0,Y 270.345,Z 550.799,A -85,B 0,C 180,E1 -17626.787,E2 -17626.787} C_VEL
LIN {X 0,Y 270.541,Z 550.78,A -85,B 0,C 180,E1 -17631.033,E2 -17631.033} C_VEL
LIN {X 0,Y 270.533,Z 550.782,A -85,B 0,C 180,E1 -17634.035,E2 -17634.035} C_VEL
LIN {X 0,Y 270.782,Z 550.745,A -85,B 0,C 180,E1 -17638.513,E2 -17638.513} C_VEL
LIN {X 0,Y 270.782,Z 550.752,A -85,B 0,C 180,E1 -17641.487,E2 -17641.487} C_VEL
LIN {X 0,Y 270.592,Z 550.773,A -85,B 0,C 180,E1 -17647.462,E2 -17647.462} C_VEL
LIN {X 0,Y 270.407,Z 550.8,A -85,B 0,C 180,E1 -17650.482,E2 -17650.482} C_VEL
LIN {X 0,Y 270.39,Z 550.802,A -85,B 0,C 180,E1 -17655.065,E2 -17655.065} C_VEL
LIN {X 0,Y 270.295,Z 550.813,A -85,B 0,C 180,E1 -17659.756,E2 -17659.756} C_VEL
LIN {X 0,Y 270.233,Z 550.822,A -85,B 0,C 180,E1 -17664.59,E2 -17664.59} C_VEL
LIN {X 0,Y 270.267,Z 550.811,A -85,B 0,C 180,E1 -17667.909,E2 -17667.909} C_VEL
LIN {X 0,Y 270.18,Z 550.829,A -85,B 0,C 180,E1 -17671.349,E2 -17671.349} C_VEL
LIN {X 0,Y 270.211,Z 550.828,A -85,B 0,C 180,E1 -17674.904,E2 -17674.904} C_VEL
LIN {X 0,Y 270.219,Z 550.827,A -85,B 0,C 180,E1 -17678.718,E2 -17678.718} C_VEL
LIN {X 0,Y 270.192,Z 550.83,A -85,B 0,C 180,E1 -17682.554,E2 -17682.554} C_VEL
LIN {X 0,Y 270.169,Z 550.833,A -85,B 0,C 180,E1 -17686.75,E2 -17686.75} C_VEL
LIN {X 0,Y 270.195,Z 550.83,A -85,B 0,C 180,E1 -17691.29,E2 -17691.29} C_VEL
LIN {X 0,Y 270.257,Z 551.02,A -85,B 0,C 180,E1 -17691.74,E2 -17691.74} C_VEL
LIN {X 0,Y 272.574,Z 560.256,A -85,B 0,C 180,E1 -17695.597,E2 -17695.597} C_VEL
LIN {X 0,Y 274.316,Z 567.926,A -85,B 0,C 180,E1 -17698.593,E2 -17698.593} C_VEL
LIN {X 0,Y 282.757,Z 586.989,A -85,B 0,C 180,E1 -17700.254,E2 -17700.254} C_VEL
LIN {X 0,Y 283.754,Z 590.111,A -85,B 0,C 180,E1 -17700.467,E2 -17700.467} C_VEL
LIN {X 0,Y 288.025,Z 615.315,A -85,B 0,C 180,E1 -17701.691,E2 -17701.691} C_VEL
LIN {X 0,Y 286.034,Z 676.797,A -85,B 0,C 180,E1 -17703.24,E2 -17703.24} C_VEL
LIN {X 0,Y 284.961,Z 690.167,A -85,B 0,C 180,E1 -17703.842,E2 -17703.842} C_VEL
LIN {X 0,Y 283.391,Z 702.699,A -85,B 0,C 180,E1 -17704.673,E2 -17704.673} C_VEL
LIN {X 0,Y 281.793,Z 713.85,A -85,B 0,C 180,E1 -17705.701,E2 -17705.701} C_VEL
LIN {X 0,Y 279.659,Z 725.436,A -85,B 0,C 180,E1 -17707.076,E2 -17707.076} C_VEL
LIN {X 0,Y 277.503,Z 735.87,A -85,B 0,C 180,E1 -17708.651,E2 -17708.651} C_VEL
LIN {X 0,Y 275.645,Z 744.407,A -85,B 0,C 180,E1 -17710.256,E2 -17710.256} C_VEL
LIN {X 0,Y 273.914,Z 752.291,A -85,B 0,C 180,E1 -17712.068,E2 -17712.068} C_VEL
LIN {X 0,Y 272.112,Z 760.01,A -85,B 0,C 180,E1 -17714.265,E2 -17714.265} C_VEL
LIN {X 0,Y 270.532,Z 766.214,A -85,B 0,C 180,E1 -17716.479,E2 -17716.479} C_VEL
LIN {X 0,Y 269.522,Z 771.158,A -85,B 0,C 180,E1 -17718.722,E2 -17718.722} C_VEL
LIN {X 0,Y 268.775,Z 774.984,A -85,B 0,C 180,E1 -17720.974,E2 -17720.974} C_VEL
LIN {X 0,Y 268.45,Z 776.962,A -85,B 0,C 180,E1 -17722.479,E2 -17722.479} C_VEL
LIN {X 0,Y 268.171,Z 779.174,A -85,B 0,C 180,E1 -17724.793,E2 -17724.793} C_VEL
LIN {X 0,Y 268.167,Z 780.387,A -85,B 0,C 180,E1 -17726.996,E2 -17726.996} C_VEL
LIN {X 0,Y 268.188,Z 780.721,A -85,B 0,C 180,E1 -17728.498,E2 -17728.498} C_VEL
LIN {X 0,Y 268.202,Z 780.669,A -85,B 0,C 180,E1 -17730,E2 -17730} C_VEL
LIN {X 0,Y 268.189,Z 780.207,A -85,B 0,C 180,E1 -17731.502,E2 -17731.502} C_VEL
LIN {X 0,Y 268.168,Z 779.315,A -85,B 0,C 180,E1 -17733.004,E2 -17733.004} C_VEL
LIN {X 0,Y 268.216,Z 777.173,A -85,B 0,C 180,E1 -17735.312,E2 -17735.312} C_VEL
LIN {X 0,Y 268.415,Z 774.167,A -85,B 0,C 180,E1 -17737.522,E2 -17737.522} C_VEL
LIN {X 0,Y 268.894,Z 770.04,A -85,B 0,C 180,E1 -17739.781,E2 -17739.781} C_VEL
LIN {X 0,Y 269.763,Z 763.715,A -85,B 0,C 180,E1 -17742.411,E2 -17742.411} C_VEL
LIN {X 0,Y 271.03,Z 756.835,A -85,B 0,C 180,E1 -17744.644,E2 -17744.644} C_VEL
LIN {X 0,Y 272.594,Z 748.36,A -85,B 0,C 180,E1 -17746.831,E2 -17746.831} C_VEL
LIN {X 0,Y 274.028,Z 739.389,A -85,B 0,C 180,E1 -17748.697,E2 -17748.697} C_VEL
LIN {X 0,Y 275.788,Z 728.494,A -85,B 0,C 180,E1 -17750.511,E2 -17750.511} C_VEL
LIN {X 0,Y 277.486,Z 717.538,A -85,B 0,C 180,E1 -17751.936,E2 -17751.936} C_VEL
LIN {X 0,Y 279.059,Z 705.231,A -85,B 0,C 180,E1 -17753.172,E2 -17753.172} C_VEL
LIN {X 0,Y 280.484,Z 692.273,A -85,B 0,C 180,E1 -17754.125,E2 -17754.125} C_VEL
LIN {X 0,Y 281.471,Z 679.097,A -85,B 0,C 180,E1 -17754.771,E2 -17754.771} C_VEL
LIN {X 0,Y 282.158,Z 659.07,A -85,B 0,C 180,E1 -17755.332,E2 -17755.332} C_VEL
LIN {X 0,Y 283.272,Z 613.296,A -85,B 0,C 180,E1 -17756.479,E2 -17756.479} C_VEL
LIN {X 0,Y 279.534,Z 586.772,A -85,B 0,C 180,E1 -17757.567,E2 -17757.567} C_VEL
LIN {X 0,Y 277.793,Z 578.124,A -85,B 0,C 180,E1 -17757.983,E2 -17757.983} C_VEL
LIN {X 0,Y 273.988,Z 568.191,A -85,B 0,C 180,E1 -17758.673,E2 -17758.673} C_VEL
LIN {X 0,Y 271.792,Z 557.576,A -85,B 0,C 180,E1 -17762.519,E2 -17762.519} C_VEL
LIN {X 0,Y 270.249,Z 550.82,A -85,B 0,C 180,E1 -17765.125,E2 -17765.125} C_VEL
LIN {X 0,Y 270.22,Z 550.825,A -85,B 0,C 180,E1 -17768.716,E2 -17768.716} C_VEL
LIN {X 0,Y 270.169,Z 550.832,A -85,B 0,C 180,E1 -17773.25,E2 -17773.25} C_VEL
LIN {X 0,Y 270.192,Z 550.829,A -85,B 0,C 180,E1 -17777.446,E2 -17777.446} C_VEL
LIN {X 0,Y 270.241,Z 550.824,A -85,B 0,C 180,E1 -17781.38,E2 -17781.38} C_VEL
LIN {X 0,Y 270.211,Z 550.826,A -85,B 0,C 180,E1 -17785.096,E2 -17785.096} C_VEL
LIN {X 0,Y 270.196,Z 550.827,A -85,B 0,C 180,E1 -17789.13,E2 -17789.13} C_VEL
LIN {X 0,Y 270.26,Z 550.815,A -85,B 0,C 180,E1 -17792.145,E2 -17792.145} C_VEL
LIN {X 0,Y 270.232,Z 550.822,A -85,B 0,C 180,E1 -17795.537,E2 -17795.537} C_VEL
LIN {X 0,Y 270.294,Z 550.814,A -85,B 0,C 180,E1 -17800.244,E2 -17800.244} C_VEL
LIN {X 0,Y 270.39,Z 550.802,A -85,B 0,C 180,E1 -17804.935,E2 -17804.935} C_VEL
LIN {X 0,Y 270.435,Z 550.794,A -85,B 0,C 180,E1 -17809.519,E2 -17809.519} C_VEL
LIN {X 0,Y 270.602,Z 550.776,A -85,B 0,C 180,E1 -17812.539,E2 -17812.539} C_VEL
LIN {X 0,Y 270.781,Z 550.753,A -85,B 0,C 180,E1 -17818.513,E2 -17818.513} C_VEL
LIN {X 0,Y 270.781,Z 550.75,A -85,B 0,C 180,E1 -17821.487,E2 -17821.487} C_VEL
LIN {X 0,Y 270.593,Z 550.778,A -85,B 0,C 180,E1 -17827.462,E2 -17827.462} C_VEL
LIN {X 0,Y 270.407,Z 550.788,A -85,B 0,C 180,E1 -17830.483,E2 -17830.483} C_VEL
LIN {X 0,Y 270.391,Z 550.803,A -85,B 0,C 180,E1 -17835.066,E2 -17835.066} C_VEL
LIN {X 0,Y 270.297,Z 550.804,A -85,B 0,C 180,E1 -17839.756,E2 -17839.756} C_VEL
LIN {X 0,Y 270.27,Z 550.817,A -85,B 0,C 180,E1 -17844.586,E2 -17844.586} C_VEL
LIN {X 0,Y 270.268,Z 550.818,A -85,B 0,C 180,E1 -17847.909,E2 -17847.909} C_VEL
LIN {X 0,Y 270.181,Z 550.828,A -85,B 0,C 180,E1 -17851.349,E2 -17851.349} C_VEL
LIN {X 0,Y 270.211,Z 550.825,A -85,B 0,C 180,E1 -17854.905,E2 -17854.905} C_VEL
LIN {X 0,Y 270.195,Z 550.819,A -85,B 0,C 180,E1 -17858.711,E2 -17858.711} C_VEL
LIN {X 0,Y 270.192,Z 550.826,A -85,B 0,C 180,E1 -17862.555,E2 -17862.555} C_VEL
LIN {X 0,Y 270.211,Z 550.823,A -85,B 0,C 180,E1 -17866.741,E2 -17866.741} C_VEL
LIN {X 0,Y 270.245,Z 550.822,A -85,B 0,C 180,E1 -17869.448,E2 -17869.448} C_VEL
LIN {X 0,Y 270.257,Z 550.82,A -85,B 0,C 180,E1 -17873.722,E2 -17873.722} C_VEL
LIN {X 0,Y 270.205,Z 550.828,A -85,B 0,C 180,E1 -17876.894,E2 -17876.894} C_VEL
LIN {X 0,Y 270.23,Z 550.826,A -85,B 0,C 180,E1 -17880.388,E2 -17880.388} C_VEL
LIN {X 0,Y 270.328,Z 550.838,A -85,B 0,C 180,E1 -17883.46,E2 -17883.46} C_VEL
LIN {X 0,Y 271.199,Z 554.82,A -85,B 0,C 180,E1 -17885.096,E2 -17885.096} C_VEL
LIN {X 0,Y 280.536,Z 577.533,A -85,B 0,C 180,E1 -17886.731,E2 -17886.731} C_VEL
LIN {X 0,Y 283.237,Z 585.608,A -85,B 0,C 180,E1 -17887.216,E2 -17887.216} C_VEL
LIN {X 0,Y 283.976,Z 590.288,A -85,B 0,C 180,E1 -17887.415,E2 -17887.415} C_VEL
LIN {X 0,Y 281.964,Z 661.54,A -85,B 0,C 180,E1 -17889.211,E2 -17889.211} C_VEL
LIN {X 0,Y 281.209,Z 674.496,A -85,B 0,C 180,E1 -17889.806,E2 -17889.806} C_VEL
LIN {X 0,Y 280.203,Z 686.097,A -85,B 0,C 180,E1 -17890.59,E2 -17890.59} C_VEL
LIN {X 0,Y 278.864,Z 697.68,A -85,B 0,C 180,E1 -17891.638,E2 -17891.638} C_VEL
LIN {X 0,Y 277.281,Z 709.524,A -85,B 0,C 180,E1 -17893.054,E2 -17893.054} C_VEL
LIN {X 0,Y 275.618,Z 720.078,A -85,B 0,C 180,E1 -17894.66,E2 -17894.66} C_VEL
LIN {X 0,Y 273.957,Z 728.718,A -85,B 0,C 180,E1 -17896.273,E2 -17896.273} C_VEL
LIN {X 0,Y 272.708,Z 736.649,A -85,B 0,C 180,E1 -17898.102,E2 -17898.102} C_VEL
LIN {X 0,Y 271.337,Z 744.441,A -85,B 0,C 180,E1 -17900.308,E2 -17900.308} C_VEL
LIN {X 0,Y 270.225,Z 750.665,A -85,B 0,C 180,E1 -17902.528,E2 -17902.528} C_VEL
LIN {X 0,Y 269.346,Z 755.624,A -85,B 0,C 180,E1 -17904.76,E2 -17904.76} C_VEL
LIN {X 0,Y 268.624,Z 759.471,A -85,B 0,C 180,E1 -17907.001,E2 -17907.001} C_VEL
LIN {X 0,Y 268.395,Z 761.45,A -85,B 0,C 180,E1 -17908.5,E2 -17908.5} C_VEL
LIN {X 0,Y 268.255,Z 763.019,A -85,B 0,C 180,E1 -17910,E2 -17910} C_VEL
LIN {X 0,Y 268.222,Z 764.18,A -85,B 0,C 180,E1 -17911.501,E2 -17911.501} C_VEL
LIN {X 0,Y 268.205,Z 764.908,A -85,B 0,C 180,E1 -17913.004,E2 -17913.004} C_VEL
LIN {X 0,Y 268.224,Z 765.296,A -85,B 0,C 180,E1 -17915.325,E2 -17915.325} C_VEL
LIN {X 0,Y 268.296,Z 764.81,A -85,B 0,C 180,E1 -17917.526,E2 -17917.526} C_VEL
LIN {X 0,Y 268.456,Z 763.958,A -85,B 0,C 180,E1 -17919.037,E2 -17919.037} C_VEL
LIN {X 0,Y 269.066,Z 761.06,A -85,B 0,C 180,E1 -17922.061,E2 -17922.061} C_VEL
LIN {X 0,Y 269.902,Z 757.729,A -85,B 0,C 180,E1 -17924.322,E2 -17924.322} C_VEL
LIN {X 0,Y 270.974,Z 753.315,A -85,B 0,C 180,E1 -17926.576,E2 -17926.576} C_VEL
LIN {X 0,Y 272.652,Z 746.601,A -85,B 0,C 180,E1 -17929.186,E2 -17929.186} C_VEL
LIN {X 0,Y 274.503,Z 739.261,A -85,B 0,C 180,E1 -17931.397,E2 -17931.397} C_VEL
LIN {X 0,Y 276.514,Z 730.644,A -85,B 0,C 180,E1 -17933.473,E2 -17933.473} C_VEL
LIN {X 0,Y 278.653,Z 720.594,A -85,B 0,C 180,E1 -17935.388,E2 -17935.388} C_VEL
LIN {X 0,Y 280.741,Z 709.998,A -85,B 0,C 180,E1 -17936.983,E2 -17936.983} C_VEL
LIN {X 0,Y 282.504,Z 699.761,A -85,B 0,C 180,E1 -17938.207,E2 -17938.207} C_VEL
LIN {X 0,Y 284.202,Z 687.617,A -85,B 0,C 180,E1 -17939.336,E2 -17939.336} C_VEL
LIN {X 0,Y 285.47,Z 675.358,A -85,B 0,C 180,E1 -17940.17,E2 -17940.17} C_VEL
LIN {X 0,Y 286.42,Z 662.598,A -85,B 0,C 180,E1 -17940.754,E2 -17940.754} C_VEL
LIN {X 0,Y 288.764,Z 593.863,A -85,B 0,C 180,E1 -17942.474,E2 -17942.474} C_VEL
LIN {X 0,Y 288.221,Z 591.757,A -85,B 0,C 180,E1 -17942.597,E2 -17942.597} C_VEL
LIN {X 0,Y 281.145,Z 575.129,A -85,B 0,C 180,E1 -17943.94,E2 -17943.94} C_VEL
LIN {X 0,Y 272.852,Z 558.469,A -85,B 0,C 180,E1 -17945.544,E2 -17945.544} C_VEL
LIN {X 0,Y 271.278,Z 555.097,A -85,B 0,C 180,E1 -17945.913,E2 -17945.913} C_VEL
LIN {X 0,Y 270.25,Z 550.817,A -85,B 0,C 180,E1 -17947.906,E2 -17947.906} C_VEL
LIN {X 0,Y 270.248,Z 550.823,A -85,B 0,C 180,E1 -17951.047,E2 -17951.047} C_VEL
LIN {X 0,Y 270.194,Z 550.826,A -85,B 0,C 180,E1 -17955.388,E2 -17955.388} C_VEL
LIN {X 0,Y 270.211,Z 550.81,A -85,B 0,C 180,E1 -17959.44,E2 -17959.44} C_VEL
LIN {X 0,Y 270.254,Z 550.818,A -85,B 0,C 180,E1 -17963.72,E2 -17963.72} C_VEL
LIN {X 0,Y 270.201,Z 550.825,A -85,B 0,C 180,E1 -17966.892,E2 -17966.892} C_VEL
LIN {X 0,Y 270.225,Z 550.819,A -85,B 0,C 180,E1 -17970.386,E2 -17970.386} C_VEL
LIN {X 0,Y 270.259,Z 550.812,A -85,B 0,C 180,E1 -17973.763,E2 -17973.763} C_VEL
LIN {X 0,Y 270.228,Z 550.816,A -85,B 0,C 180,E1 -17977.038,E2 -17977.038} C_VEL
LIN {X 0,Y 270.292,Z 550.816,A -85,B 0,C 180,E1 -17980.301,E2 -17980.301} C_VEL
LIN {X 0,Y 270.397,Z 550.803,A -85,B 0,C 180,E1 -17984.935,E2 -17984.935} C_VEL
LIN {X 0,Y 270.345,Z 550.799,A -85,B 0,C 180,E1 -17986.787,E2 -17986.787} C_VEL
LIN {X 0,Y 269.695,Z 550.882,A -85,B 0,C 180,E1 -17988.032,E2 -17988.032} C_VEL
LIN {X 0,Y 266.928,Z 551.235,A -85,B 0,C 180,E1 -17990.063,E2 -17990.063} C_VEL
LIN {X 0,Y 264.583,Z 551.52,A -85,B 0,C 180,E1 -17991.714,E2 -17991.714} C_VEL
LIN {X 0,Y 263.579,Z 551.643,A -85,B 0,C 180,E1 -17992.992,E2 -17992.992} C_VEL
LIN {X 0,Y 263.498,Z 551.653,A -85,B 0,C 180,E1 -17993.424,E2 -17993.424} C_VEL
LIN {X 0,Y 263.746,Z 551.62,A -85,B 0,C 180,E1 -17998.473,E2 -17998.473} C_VEL
LIN {X 0,Y 263.746,Z 551.629,A -85,B 0,C 180,E1 -18001.527,E2 -18001.527} C_VEL
LIN {X 0,Y 263.552,Z 551.649,A -85,B 0,C 180,E1 -18007.662,E2 -18007.662} C_VEL
LIN {X 0,Y 263.349,Z 551.682,A -85,B 0,C 180,E1 -18010.766,E2 -18010.766} C_VEL
LIN {X 0,Y 263.339,Z 551.681,A -85,B 0,C 180,E1 -18015.479,E2 -18015.479} C_VEL
LIN {X 0,Y 263.257,Z 551.692,A -85,B 0,C 180,E1 -18020.307,E2 -18020.307} C_VEL
LIN {X 0,Y 263.188,Z 551.7,A -85,B 0,C 180,E1 -18025.293,E2 -18025.293} C_VEL
LIN {X 0,Y 263.175,Z 551.701,A -85,B 0,C 180,E1 -18028.73,E2 -18028.73} C_VEL
LIN {X 0,Y 263.129,Z 551.708,A -85,B 0,C 180,E1 -18032.289,E2 -18032.289} C_VEL
LIN {X 0,Y 263.184,Z 551.701,A -85,B 0,C 180,E1 -18035.978,E2 -18035.978} C_VEL
LIN {X 0,Y 263.15,Z 551.706,A -85,B 0,C 180,E1 -18039.864,E2 -18039.864} C_VEL
LIN {X 0,Y 263.131,Z 551.71,A -85,B 0,C 180,E1 -18043.982,E2 -18043.982} C_VEL
LIN {X 0,Y 263.122,Z 551.711,A -85,B 0,C 180,E1 -18048.407,E2 -18048.407} C_VEL
LIN {X 0,Y 263.151,Z 551.862,A -85,B 0,C 180,E1 -18050.867,E2 -18050.867} C_VEL
LIN {X 0,Y 265.22,Z 559.8,A -85,B 0,C 180,E1 -18054.341,E2 -18054.341} C_VEL
LIN {X 0,Y 267.021,Z 567.651,A -85,B 0,C 180,E1 -18057.553,E2 -18057.553} C_VEL
LIN {X 0,Y 274.907,Z 584.867,A -85,B 0,C 180,E1 -18059.188,E2 -18059.188} C_VEL
LIN {X 0,Y 277.777,Z 591.865,A -85,B 0,C 180,E1 -18059.772,E2 -18059.772} C_VEL
LIN {X 0,Y 281.914,Z 616.71,A -85,B 0,C 180,E1 -18061.015,E2 -18061.015} C_VEL
LIN {X 0,Y 279.803,Z 676.716,A -85,B 0,C 180,E1 -18062.55,E2 -18062.55} C_VEL
LIN {X 0,Y 278.623,Z 690.719,A -85,B 0,C 180,E1 -18063.201,E2 -18063.201} C_VEL
LIN {X 0,Y 277.013,Z 703.02,A -85,B 0,C 180,E1 -18064.047,E2 -18064.047} C_VEL
LIN {X 0,Y 275.354,Z 714.036,A -85,B 0,C 180,E1 -18065.094,E2 -18065.094} C_VEL
LIN {X 0,Y 273.151,Z 725.55,A -85,B 0,C 180,E1 -18066.497,E2 -18066.497} C_VEL
LIN {X 0,Y 270.909,Z 735.929,A -85,B 0,C 180,E1 -18068.105,E2 -18068.105} C_VEL
LIN {X 0,Y 268.952,Z 744.422,A -85,B 0,C 180,E1 -18069.743,E2 -18069.743} C_VEL
LIN {X 0,Y 267.152,Z 752.268,A -85,B 0,C 180,E1 -18071.598,E2 -18071.598} C_VEL
LIN {X 0,Y 265.277,Z 759.943,A -85,B 0,C 180,E1 -18073.849,E2 -18073.849} C_VEL
LIN {X 0,Y 263.616,Z 766.12,A -85,B 0,C 180,E1 -18076.117,E2 -18076.117} C_VEL
LIN {X 0,Y 262.524,Z 771.04,A -85,B 0,C 180,E1 -18078.418,E2 -18078.418} C_VEL
LIN {X 0,Y 261.744,Z 774.844,A -85,B 0,C 180,E1 -18080.729,E2 -18080.729} C_VEL
LIN {X 0,Y 261.154,Z 778.37,A -85,B 0,C 180,E1 -18083.821,E2 -18083.821} C_VEL
LIN {X 0,Y 261.066,Z 779.487,A -85,B 0,C 180,E1 -18085.368,E2 -18085.368} C_VEL
LIN {X 0,Y 261.063,Z 780.197,A -85,B 0,C 180,E1 -18086.914,E2 -18086.914} C_VEL
LIN {X 0,Y 261.115,Z 780.522,A -85,B 0,C 180,E1 -18088.458,E2 -18088.458} C_VEL
LIN {X 0,Y 261.128,Z 780.46,A -85,B 0,C 180,E1 -18090,E2 -18090} C_VEL
LIN {X 0,Y 261.116,Z 779.979,A -85,B 0,C 180,E1 -18091.542,E2 -18091.542} C_VEL
LIN {X 0,Y 261.083,Z 779.076,A -85,B 0,C 180,E1 -18093.086,E2 -18093.086} C_VEL
LIN {X 0,Y 261.131,Z 777.154,A -85,B 0,C 180,E1 -18095.249,E2 -18095.249} C_VEL
LIN {X 0,Y 261.349,Z 773.885,A -85,B 0,C 180,E1 -18097.727,E2 -18097.727} C_VEL
LIN {X 0,Y 261.853,Z 769.734,A -85,B 0,C 180,E1 -18100.047,E2 -18100.047} C_VEL
LIN {X 0,Y 262.804,Z 763.385,A -85,B 0,C 180,E1 -18102.745,E2 -18102.745} C_VEL
LIN {X 0,Y 264.149,Z 756.477,A -85,B 0,C 180,E1 -18105.035,E2 -18105.035} C_VEL
LIN {X 0,Y 265.486,Z 749.417,A -85,B 0,C 180,E1 -18106.929,E2 -18106.929} C_VEL
LIN {X 0,Y 266.94,Z 740.895,A -85,B 0,C 180,E1 -18108.815,E2 -18108.815} C_VEL
LIN {X 0,Y 268.517,Z 731.539,A -85,B 0,C 180,E1 -18110.491,E2 -18110.491} C_VEL
LIN {X 0,Y 270.41,Z 719.932,A -85,B 0,C 180,E1 -18112.139,E2 -18112.139} C_VEL
LIN {X 0,Y 272.056,Z 708.487,A -85,B 0,C 180,E1 -18113.401,E2 -18113.401} C_VEL
LIN {X 0,Y 273.453,Z 696.68,A -85,B 0,C 180,E1 -18114.382,E2 -18114.382} C_VEL
LIN {X 0,Y 274.694,Z 683.047,A -85,B 0,C 180,E1 -18115.172,E2 -18115.172} C_VEL
LIN {X 0,Y 275.299,Z 670.856,A -85,B 0,C 180,E1 -18115.619,E2 -18115.619} C_VEL
LIN {X 0,Y 276.856,Z 614.28,A -85,B 0,C 180,E1 -18117.058,E2 -18117.058} C_VEL
LIN {X 0,Y 273.106,Z 587.629,A -85,B 0,C 180,E1 -18118.19,E2 -18118.19} C_VEL
LIN {X 0,Y 271.704,Z 580.852,A -85,B 0,C 180,E1 -18118.532,E2 -18118.532} C_VEL
LIN {X 0,Y 266.72,Z 567.971,A -85,B 0,C 180,E1 -18119.469,E2 -18119.469} C_VEL
LIN {X 0,Y 264.799,Z 558.646,A -85,B 0,C 180,E1 -18122.961,E2 -18122.961} C_VEL
LIN {X 0,Y 263.253,Z 551.689,A -85,B 0,C 180,E1 -18125.744,E2 -18125.744} C_VEL
LIN {X 0,Y 263.113,Z 551.71,A -85,B 0,C 180,E1 -18129.87,E2 -18129.87} C_VEL
LIN {X 0,Y 263.126,Z 551.707,A -85,B 0,C 180,E1 -18133.982,E2 -18133.982} C_VEL
LIN {X 0,Y 263.145,Z 551.705,A -85,B 0,C 180,E1 -18138.4,E2 -18138.4} C_VEL
LIN {X 0,Y 263.184,Z 551.7,A -85,B 0,C 180,E1 -18142.107,E2 -18142.107} C_VEL
LIN {X 0,Y 263.18,Z 551.7,A -85,B 0,C 180,E1 -18145.89,E2 -18145.89} C_VEL
LIN {X 0,Y 263.147,Z 551.708,A -85,B 0,C 180,E1 -18149.506,E2 -18149.506} C_VEL
LIN {X 0,Y 263.187,Z 551.697,A -85,B 0,C 180,E1 -18153.002,E2 -18153.002} C_VEL
LIN {X 0,Y 263.149,Z 551.7,A -85,B 0,C 180,E1 -18156.384,E2 -18156.384} C_VEL
LIN {X 0,Y 263.257,Z 551.693,A -85,B 0,C 180,E1 -18159.693,E2 -18159.693} C_VEL
LIN {X 0,Y 263.339,Z 551.68,A -85,B 0,C 180,E1 -18164.521,E2 -18164.521} C_VEL
LIN {X 0,Y 263.368,Z 551.672,A -85,B 0,C 180,E1 -18169.234,E2 -18169.234} C_VEL
LIN {X 0,Y 263.564,Z 551.652,A -85,B 0,C 180,E1 -18172.338,E2 -18172.338} C_VEL
LIN {X 0,Y 263.745,Z 551.63,A -85,B 0,C 180,E1 -18178.473,E2 -18178.473} C_VEL
LIN {X 0,Y 263.745,Z 551.625,A -85,B 0,C 180,E1 -18181.527,E2 -18181.527} C_VEL
LIN {X 0,Y 263.552,Z 551.653,A -85,B 0,C 180,E1 -18187.662,E2 -18187.662} C_VEL
LIN {X 0,Y 263.349,Z 551.666,A -85,B 0,C 180,E1 -18190.767,E2 -18190.767} C_VEL
LIN {X 0,Y 263.339,Z 551.684,A -85,B 0,C 180,E1 -18195.479,E2 -18195.479} C_VEL
LIN {X 0,Y 263.26,Z 551.679,A -85,B 0,C 180,E1 -18200.307,E2 -18200.307} C_VEL
LIN {X 0,Y 263.204,Z 551.7,A -85,B 0,C 180,E1 -18205.292,E2 -18205.292} C_VEL
LIN {X 0,Y 263.176,Z 551.701,A -85,B 0,C 180,E1 -18208.73,E2 -18208.73} C_VEL
LIN {X 0,Y 263.13,Z 551.705,A -85,B 0,C 180,E1 -18212.289,E2 -18212.289} C_VEL
LIN {X 0,Y 263.183,Z 551.694,A -85,B 0,C 180,E1 -18215.979,E2 -18215.979} C_VEL
LIN {X 0,Y 263.109,Z 551.71,A -85,B 0,C 180,E1 -18219.872,E2 -18219.872} C_VEL
LIN {X 0,Y 263.137,Z 551.707,A -85,B 0,C 180,E1 -18223.982,E2 -18223.982} C_VEL
LIN {X 0,Y 263.172,Z 551.7,A -85,B 0,C 180,E1 -18228.395,E2 -18228.395} C_VEL
LIN {X 0,Y 263.189,Z 551.699,A -85,B 0,C 180,E1 -18232.109,E2 -18232.109} C_VEL
LIN {X 0,Y 263.184,Z 551.701,A -85,B 0,C 180,E1 -18235.891,E2 -18235.891} C_VEL
LIN {X 0,Y 263.152,Z 551.708,A -85,B 0,C 180,E1 -18239.508,E2 -18239.508} C_VEL
LIN {X 0,Y 263.295,Z 551.808,A -85,B 0,C 180,E1 -18242.92,E2 -18242.92} C_VEL
LIN {X 0,Y 264.09,Z 555.328,A -85,B 0,C 180,E1 -18244.328,E2 -18244.328} C_VEL
LIN {X 0,Y 272.617,Z 575.418,A -85,B 0,C 180,E1 -18245.864,E2 -18245.864} C_VEL
LIN {X 0,Y 276.832,Z 586.834,A -85,B 0,C 180,E1 -18246.623,E2 -18246.623} C_VEL
LIN {X 0,Y 277.522,Z 591.632,A -85,B 0,C 180,E1 -18246.827,E2 -18246.827} C_VEL
LIN {X 0,Y 275.423,Z 662.109,A -85,B 0,C 180,E1 -18248.645,E2 -18248.645} C_VEL
LIN {X 0,Y 274.572,Z 675.682,A -85,B 0,C 180,E1 -18249.296,E2 -18249.296} C_VEL
LIN {X 0,Y 273.451,Z 688.144,A -85,B 0,C 180,E1 -18250.189,E2 -18250.189} C_VEL
LIN {X 0,Y 271.961,Z 700.047,A -85,B 0,C 180,E1 -18251.35,E2 -18251.35} C_VEL
LIN {X 0,Y 270.345,Z 711.424,A -85,B 0,C 180,E1 -18252.8,E2 -18252.8} C_VEL
LIN {X 0,Y 268.615,Z 721.688,A -85,B 0,C 180,E1 -18254.444,E2 -18254.444} C_VEL
LIN {X 0,Y 266.771,Z 730.921,A -85,B 0,C 180,E1 -18256.285,E2 -18256.285} C_VEL
LIN {X 0,Y 265.243,Z 740.162,A -85,B 0,C 180,E1 -18258.63,E2 -18258.63} C_VEL
LIN {X 0,Y 263.924,Z 747.044,A -85,B 0,C 180,E1 -18260.806,E2 -18260.806} C_VEL
LIN {X 0,Y 262.874,Z 752.809,A -85,B 0,C 180,E1 -18263.09,E2 -18263.09} C_VEL
LIN {X 0,Y 261.96,Z 757.358,A -85,B 0,C 180,E1 -18265.384,E2 -18265.384} C_VEL
LIN {X 0,Y 261.559,Z 759.761,A -85,B 0,C 180,E1 -18266.92,E2 -18266.92} C_VEL
LIN {X 0,Y 261.319,Z 761.725,A -85,B 0,C 180,E1 -18268.459,E2 -18268.459} C_VEL
LIN {X 0,Y 261.178,Z 763.281,A -85,B 0,C 180,E1 -18270,E2 -18270} C_VEL
LIN {X 0,Y 261.148,Z 764.418,A -85,B 0,C 180,E1 -18271.542,E2 -18271.542} C_VEL
LIN {X 0,Y 261.117,Z 765.132,A -85,B 0,C 180,E1 -18273.086,E2 -18273.086} C_VEL
LIN {X 0,Y 261.139,Z 765.426,A -85,B 0,C 180,E1 -18276.18,E2 -18276.18} C_VEL
LIN {X 0,Y 261.238,Z 764.987,A -85,B 0,C 180,E1 -18277.73,E2 -18277.73} C_VEL
LIN {X 0,Y 261.691,Z 762.856,A -85,B 0,C 180,E1 -18280.835,E2 -18280.835} C_VEL
LIN {X 0,Y 262.374,Z 760.172,A -85,B 0,C 180,E1 -18283.16,E2 -18283.16} C_VEL
LIN {X 0,Y 263.317,Z 756.465,A -85,B 0,C 180,E1 -18285.48,E2 -18285.48} C_VEL
LIN {X 0,Y 264.541,Z 751.627,A -85,B 0,C 180,E1 -18287.789,E2 -18287.789} C_VEL
LIN {X 0,Y 266.186,Z 745.509,A -85,B 0,C 180,E1 -18290.074,E2 -18290.074} C_VEL
LIN {X 0,Y 268.232,Z 737.881,A -85,B 0,C 180,E1 -18292.328,E2 -18292.328} C_VEL
LIN {X 0,Y 270.069,Z 729.941,A -85,B 0,C 180,E1 -18294.219,E2 -18294.219} C_VEL
LIN {X 0,Y 272.391,Z 719.378,A -85,B 0,C 180,E1 -18296.221,E2 -18296.221} C_VEL
LIN {X 0,Y 274.619,Z 708.468,A -85,B 0,C 180,E1 -18297.842,E2 -18297.842} C_VEL
LIN {X 0,Y 276.544,Z 697.756,A -85,B 0,C 180,E1 -18299.08,E2 -18299.08} C_VEL
LIN {X 0,Y 278.182,Z 684.812,A -85,B 0,C 180,E1 -18300.244,E2 -18300.244} C_VEL
LIN {X 0,Y 279.577,Z 672.227,A -85,B 0,C 180,E1 -18301.033,E2 -18301.033} C_VEL
LIN {X 0,Y 280.413,Z 658.724,A -85,B 0,C 180,E1 -18301.577,E2 -18301.577} C_VEL
LIN {X 0,Y 282.515,Z 594.755,A -85,B 0,C 180,E1 -18303.195,E2 -18303.195} C_VEL
LIN {X 0,Y 275.291,Z 577.748,A -85,B 0,C 180,E1 -18304.622,E2 -18304.622} C_VEL
LIN {X 0,Y 267.687,Z 562.424,A -85,B 0,C 180,E1 -18306.153,E2 -18306.153} C_VEL
LIN {X 0,Y 264.109,Z 555.326,A -85,B 0,C 180,E1 -18306.961,E2 -18306.961} C_VEL
LIN {X 0,Y 263.175,Z 551.702,A -85,B 0,C 180,E1 -18308.733,E2 -18308.733} C_VEL
LIN {X 0,Y 263.166,Z 551.703,A -85,B 0,C 180,E1 -18311.884,E2 -18311.884} C_VEL
LIN {X 0,Y 263.143,Z 551.706,A -85,B 0,C 180,E1 -18316.145,E2 -18316.145} C_VEL
LIN {X 0,Y 263.137,Z 551.697,A -85,B 0,C 180,E1 -18320.133,E2 -18320.133} C_VEL
LIN {X 0,Y 263.187,Z 551.7,A -85,B 0,C 180,E1 -18324.021,E2 -18324.021} C_VEL
LIN {X 0,Y 263.13,Z 551.708,A -85,B 0,C 180,E1 -18327.711,E2 -18327.711} C_VEL
LIN {X 0,Y 263.197,Z 551.7,A -85,B 0,C 180,E1 -18331.782,E2 -18331.782} C_VEL
LIN {X 0,Y 263.222,Z 551.697,A -85,B 0,C 180,E1 -18335.2,E2 -18335.2} C_VEL
LIN {X 0,Y 263.259,Z 551.691,A -85,B 0,C 180,E1 -18339.693,E2 -18339.693} C_VEL
LIN {X 0,Y 263.345,Z 551.682,A -85,B 0,C 180,E1 -18344.521,E2 -18344.521} C_VEL
LIN {X 0,Y 263.349,Z 551.681,A -85,B 0,C 180,E1 -18349.233,E2 -18349.233} C_VEL
LIN {X 0,Y 263.552,Z 551.645,A -85,B 0,C 180,E1 -18352.338,E2 -18352.338} C_VEL
LIN {X 0,Y 263.498,Z 551.653,A -85,B 0,C 180,E1 -18353.424,E2 -18353.424} C_VEL
LIN {X 0,Y 262.877,Z 551.74,A -85,B 0,C 180,E1 -18354.7,E2 -18354.7} C_VEL
LIN {X 0,Y 260.199,Z 552.08,A -85,B 0,C 180,E1 -18356.785,E2 -18356.785} C_VEL
LIN {X 0,Y 257.096,Z 552.461,A -85,B 0,C 180,E1 -18359.347,E2 -18359.347} C_VEL
LIN {X 0,Y 256.747,Z 552.5,A -85,B 0,C 180,E1 -18360.231,E2 -18360.231} C_VEL
LIN {X 0,Y 256.493,Z 552.522,A -85,B 0,C 180,E1 -18363.141,E2 -18363.141} C_VEL
LIN {X 0,Y 256.509,Z 552.524,A -85,B 0,C 180,E1 -18367.874,E2 -18367.874} C_VEL
LIN {X 0,Y 256.287,Z 552.552,A -85,B 0,C 180,E1 -18372.672,E2 -18372.672} C_VEL
LIN {X 0,Y 256.273,Z 552.564,A -85,B 0,C 180,E1 -18376.299,E2 -18376.299} C_VEL
LIN {X 0,Y 256.148,Z 552.577,A -85,B 0,C 180,E1 -18381.118,E2 -18381.118} C_VEL
LIN {X 0,Y 256.166,Z 552.576,A -85,B 0,C 180,E1 -18385.13,E2 -18385.13} C_VEL
LIN {X 0,Y 256.109,Z 552.582,A -85,B 0,C 180,E1 -18389.6,E2 -18389.6} C_VEL
LIN {X 0,Y 256.081,Z 552.586,A -85,B 0,C 180,E1 -18393.291,E2 -18393.291} C_VEL
LIN {X 0,Y 256.136,Z 552.579,A -85,B 0,C 180,E1 -18397.279,E2 -18397.279} C_VEL
LIN {X 0,Y 256.08,Z 552.587,A -85,B 0,C 180,E1 -18401.198,E2 -18401.198} C_VEL
LIN {X 0,Y 256.061,Z 552.59,A -85,B 0,C 180,E1 -18405.529,E2 -18405.529} C_VEL
LIN {X 0,Y 256.065,Z 552.658,A -85,B 0,C 180,E1 -18409.918,E2 -18409.918} C_VEL
LIN {X 0,Y 257.976,Z 559.746,A -85,B 0,C 180,E1 -18413.178,E2 -18413.178} C_VEL
LIN {X 0,Y 259.8,Z 567.627,A -85,B 0,C 180,E1 -18416.477,E2 -18416.477} C_VEL
LIN {X 0,Y 267.426,Z 583.548,A -85,B 0,C 180,E1 -18418.123,E2 -18418.123} C_VEL
LIN {X 0,Y 272.05,Z 594.542,A -85,B 0,C 180,E1 -18419.103,E2 -18419.103} C_VEL
LIN {X 0,Y 275.768,Z 618.086,A -85,B 0,C 180,E1 -18420.299,E2 -18420.299} C_VEL
LIN {X 0,Y 273.614,Z 676.616,A -85,B 0,C 180,E1 -18421.827,E2 -18421.827} C_VEL
LIN {X 0,Y 272.409,Z 690.52,A -85,B 0,C 180,E1 -18422.486,E2 -18422.486} C_VEL
LIN {X 0,Y 270.676,Z 703.319,A -85,B 0,C 180,E1 -18423.392,E2 -18423.392} C_VEL
LIN {X 0,Y 268.946,Z 714.229,A -85,B 0,C 180,E1 -18424.459,E2 -18424.459} C_VEL
LIN {X 0,Y 266.671,Z 725.67,A -85,B 0,C 180,E1 -18425.89,E2 -18425.89} C_VEL
LIN {X 0,Y 264.339,Z 735.992,A -85,B 0,C 180,E1 -18427.531,E2 -18427.531} C_VEL
LIN {X 0,Y 262.275,Z 744.438,A -85,B 0,C 180,E1 -18429.204,E2 -18429.204} C_VEL
LIN {X 0,Y 260.407,Z 752.241,A -85,B 0,C 180,E1 -18431.104,E2 -18431.104} C_VEL
LIN {X 0,Y 258.437,Z 759.876,A -85,B 0,C 180,E1 -18433.409,E2 -18433.409} C_VEL
LIN {X 0,Y 256.719,Z 766.027,A -85,B 0,C 180,E1 -18435.737,E2 -18435.737} C_VEL
LIN {X 0,Y 255.541,Z 770.923,A -85,B 0,C 180,E1 -18438.097,E2 -18438.097} C_VEL
LIN {X 0,Y 254.732,Z 774.705,A -85,B 0,C 180,E1 -18440.472,E2 -18440.472} C_VEL
LIN {X 0,Y 254.333,Z 776.662,A -85,B 0,C 180,E1 -18442.058,E2 -18442.058} C_VEL
LIN {X 0,Y 253.99,Z 779.157,A -85,B 0,C 180,E1 -18444.961,E2 -18444.961} C_VEL
LIN {X 0,Y 253.962,Z 780.006,A -85,B 0,C 180,E1 -18446.827,E2 -18446.827} C_VEL
LIN {X 0,Y 254.021,Z 780.322,A -85,B 0,C 180,E1 -18448.415,E2 -18448.415} C_VEL
LIN {X 0,Y 254.056,Z 780.251,A -85,B 0,C 180,E1 -18450,E2 -18450} C_VEL
LIN {X 0,Y 254.023,Z 779.749,A -85,B 0,C 180,E1 -18451.585,E2 -18451.585} C_VEL
LIN {X 0,Y 253.981,Z 778.836,A -85,B 0,C 180,E1 -18453.172,E2 -18453.172} C_VEL
LIN {X 0,Y 254.021,Z 777.195,A -85,B 0,C 180,E1 -18455.119,E2 -18455.119} C_VEL
LIN {X 0,Y 254.307,Z 773.603,A -85,B 0,C 180,E1 -18457.942,E2 -18457.942} C_VEL
LIN {X 0,Y 254.82,Z 769.427,A -85,B 0,C 180,E1 -18460.327,E2 -18460.327} C_VEL
LIN {X 0,Y 255.848,Z 763.054,A -85,B 0,C 180,E1 -18463.098,E2 -18463.098} C_VEL
LIN {X 0,Y 257.268,Z 756.118,A -85,B 0,C 180,E1 -18465.447,E2 -18465.447} C_VEL
LIN {X 0,Y 258.909,Z 747.919,A -85,B 0,C 180,E1 -18467.656,E2 -18467.656} C_VEL
LIN {X 0,Y 260.513,Z 738.486,A -85,B 0,C 180,E1 -18469.707,E2 -18469.707} C_VEL
LIN {X 0,Y 262.281,Z 728.681,A -85,B 0,C 180,E1 -18471.413,E2 -18471.413} C_VEL
LIN {X 0,Y 264.084,Z 717.922,A -85,B 0,C 180,E1 -18472.905,E2 -18472.905} C_VEL
LIN {X 0,Y 265.765,Z 705.828,A -85,B 0,C 180,E1 -18474.197,E2 -18474.197} C_VEL
LIN {X 0,Y 267.269,Z 693.213,A -85,B 0,C 180,E1 -18475.192,E2 -18475.192} C_VEL
LIN {X 0,Y 268.32,Z 680.964,A -85,B 0,C 180,E1 -18475.865,E2 -18475.865} C_VEL
LIN {X 0,Y 268.938,Z 667.148,A -85,B 0,C 180,E1 -18476.323,E2 -18476.323} C_VEL
LIN {X 0,Y 270.468,Z 615.81,A -85,B 0,C 180,E1 -18477.649,E2 -18477.649} C_VEL
LIN {X 0,Y 266.895,Z 589.583,A -85,B 0,C 180,E1 -18478.791,E2 -18478.791} C_VEL
LIN {X 0,Y 265.685,Z 583.548,A -85,B 0,C 180,E1 -18479.102,E2 -18479.102} C_VEL
LIN {X 0,Y 259.474,Z 567.692,A -85,B 0,C 180,E1 -18480.328,E2 -18480.328} C_VEL
LIN {X 0,Y 257.469,Z 558.219,A -85,B 0,C 180,E1 -18484.026,E2 -18484.026} C_VEL
LIN {X 0,Y 256.189,Z 552.571,A -85,B 0,C 180,E1 -18486.386,E2 -18486.386} C_VEL
LIN {X 0,Y 256.055,Z 552.589,A -85,B 0,C 180,E1 -18491.202,E2 -18491.202} C_VEL
LIN {X 0,Y 256.063,Z 552.589,A -85,B 0,C 180,E1 -18495.527,E2 -18495.527} C_VEL
LIN {X 0,Y 256.08,Z 552.586,A -85,B 0,C 180,E1 -18498.802,E2 -18498.802} C_VEL
LIN {X 0,Y 256.15,Z 552.576,A -85,B 0,C 180,E1 -18502.871,E2 -18502.871} C_VEL
LIN {X 0,Y 256.081,Z 552.583,A -85,B 0,C 180,E1 -18506.709,E2 -18506.709} C_VEL
LIN {X 0,Y 256.134,Z 552.576,A -85,B 0,C 180,E1 -18511.404,E2 -18511.404} C_VEL
LIN {X 0,Y 256.137,Z 552.576,A -85,B 0,C 180,E1 -18515.696,E2 -18515.696} C_VEL
LIN {X 0,Y 256.157,Z 552.576,A -85,B 0,C 180,E1 -18519.104,E2 -18519.104} C_VEL
LIN {X 0,Y 256.274,Z 552.56,A -85,B 0,C 180,E1 -18524.084,E2 -18524.084} C_VEL
LIN {X 0,Y 256.304,Z 552.551,A -85,B 0,C 180,E1 -18528.934,E2 -18528.934} C_VEL
LIN {X 0,Y 256.532,Z 552.529,A -85,B 0,C 180,E1 -18532.127,E2 -18532.127} C_VEL
LIN {X 0,Y 256.708,Z 552.506,A -85,B 0,C 180,E1 -18538.431,E2 -18538.431} C_VEL
LIN {X 0,Y 256.708,Z 552.501,A -85,B 0,C 180,E1 -18541.569,E2 -18541.569} C_VEL
LIN {X 0,Y 256.466,Z 552.534,A -85,B 0,C 180,E1 -18546.726,E2 -18546.726} C_VEL
LIN {X 0,Y 256.422,Z 552.533,A -85,B 0,C 180,E1 -18549.465,E2 -18549.465} C_VEL
LIN {X 0,Y 256.246,Z 552.563,A -85,B 0,C 180,E1 -18554.291,E2 -18554.291} C_VEL
LIN {X 0,Y 256.205,Z 552.566,A -85,B 0,C 180,E1 -18557.563,E2 -18557.563} C_VEL
LIN {X 0,Y 256.155,Z 552.566,A -85,B 0,C 180,E1 -18561.121,E2 -18561.121} C_VEL
LIN {X 0,Y 256.184,Z 552.574,A -85,B 0,C 180,E1 -18565.139,E2 -18565.139} C_VEL
LIN {X 0,Y 256.11,Z 552.583,A -85,B 0,C 180,E1 -18569.601,E2 -18569.601} C_VEL
LIN {X 0,Y 256.082,Z 552.587,A -85,B 0,C 180,E1 -18573.291,E2 -18573.291} C_VEL
LIN {X 0,Y 256.124,Z 552.569,A -85,B 0,C 180,E1 -18577.275,E2 -18577.275} C_VEL
LIN {X 0,Y 256.086,Z 552.583,A -85,B 0,C 180,E1 -18582.186,E2 -18582.186} C_VEL
LIN {X 0,Y 256.102,Z 552.581,A -85,B 0,C 180,E1 -18586.683,E2 -18586.683} C_VEL
LIN {X 0,Y 256.108,Z 552.582,A -85,B 0,C 180,E1 -18590.866,E2 -18590.866} C_VEL
LIN {X 0,Y 256.122,Z 552.581,A -85,B 0,C 180,E1 -18594.814,E2 -18594.814} C_VEL
LIN {X 0,Y 256.093,Z 552.586,A -85,B 0,C 180,E1 -18598.573,E2 -18598.573} C_VEL
LIN {X 0,Y 256.228,Z 552.637,A -85,B 0,C 180,E1 -18602.284,E2 -18602.284} C_VEL
LIN {X 0,Y 256.861,Z 555.41,A -85,B 0,C 180,E1 -18603.466,E2 -18603.466} C_VEL
LIN {X 0,Y 265.08,Z 574.397,A -85,B 0,C 180,E1 -18605.015,E2 -18605.015} C_VEL
LIN {X 0,Y 270.612,Z 588.9,A -85,B 0,C 180,E1 -18606.044,E2 -18606.044} C_VEL
LIN {X 0,Y 271.132,Z 592.897,A -85,B 0,C 180,E1 -18606.214,E2 -18606.214} C_VEL
LIN {X 0,Y 268.914,Z 662.61,A -85,B 0,C 180,E1 -18608.051,E2 -18608.051} C_VEL
LIN {X 0,Y 268.045,Z 676.097,A -85,B 0,C 180,E1 -18608.717,E2 -18608.717} C_VEL
LIN {X 0,Y 266.802,Z 689.018,A -85,B 0,C 180,E1 -18609.673,E2 -18609.673} C_VEL
LIN {X 0,Y 265.279,Z 700.754,A -85,B 0,C 180,E1 -18610.862,E2 -18610.862} C_VEL
LIN {X 0,Y 263.615,Z 712.039,A -85,B 0,C 180,E1 -18612.347,E2 -18612.347} C_VEL
LIN {X 0,Y 261.813,Z 722.226,A -85,B 0,C 180,E1 -18614.03,E2 -18614.03} C_VEL
LIN {X 0,Y 259.903,Z 731.385,A -85,B 0,C 180,E1 -18615.915,E2 -18615.915} C_VEL
LIN {X 0,Y 258.533,Z 739.361,A -85,B 0,C 180,E1 -18617.969,E2 -18617.969} C_VEL
LIN {X 0,Y 257.283,Z 745.874,A -85,B 0,C 180,E1 -18620.012,E2 -18620.012} C_VEL
LIN {X 0,Y 256.218,Z 751.363,A -85,B 0,C 180,E1 -18622.117,E2 -18622.117} C_VEL
LIN {X 0,Y 255.251,Z 756.261,A -85,B 0,C 180,E1 -18624.47,E2 -18624.47} C_VEL
LIN {X 0,Y 254.496,Z 760.05,A -85,B 0,C 180,E1 -18626.834,E2 -18626.834} C_VEL
LIN {X 0,Y 254.247,Z 762.001,A -85,B 0,C 180,E1 -18628.416,E2 -18628.416} C_VEL
LIN {X 0,Y 254.104,Z 763.543,A -85,B 0,C 180,E1 -18630,E2 -18630} C_VEL
LIN {X 0,Y 254.075,Z 764.654,A -85,B 0,C 180,E1 -18631.585,E2 -18631.585} C_VEL
LIN {X 0,Y 254.031,Z 765.356,A -85,B 0,C 180,E1 -18633.172,E2 -18633.172} C_VEL
LIN {X 0,Y 254.055,Z 765.722,A -85,B 0,C 180,E1 -18635.199,E2 -18635.199} C_VEL
LIN {X 0,Y 254.156,Z 765.161,A -85,B 0,C 180,E1 -18637.947,E2 -18637.947} C_VEL
LIN {X 0,Y 254.669,Z 763.004,A -85,B 0,C 180,E1 -18641.138,E2 -18641.138} C_VEL
LIN {X 0,Y 255.422,Z 760.291,A -85,B 0,C 180,E1 -18643.525,E2 -18643.525} C_VEL
LIN {X 0,Y 256.428,Z 756.556,A -85,B 0,C 180,E1 -18645.906,E2 -18645.906} C_VEL
LIN {X 0,Y 257.741,Z 751.687,A -85,B 0,C 180,E1 -18648.275,E2 -18648.275} C_VEL
LIN {X 0,Y 259.461,Z 745.535,A -85,B 0,C 180,E1 -18650.617,E2 -18650.617} C_VEL
LIN {X 0,Y 261.635,Z 737.855,A -85,B 0,C 180,E1 -18652.923,E2 -18652.923} C_VEL
LIN {X 0,Y 263.704,Z 729.1,A -85,B 0,C 180,E1 -18655.022,E2 -18655.022} C_VEL
LIN {X 0,Y 265.992,Z 719.241,A -85,B 0,C 180,E1 -18656.902,E2 -18656.902} C_VEL
LIN {X 0,Y 268.327,Z 708.223,A -85,B 0,C 180,E1 -18658.554,E2 -18658.554} C_VEL
LIN {X 0,Y 270.329,Z 697.397,A -85,B 0,C 180,E1 -18659.815,E2 -18659.815} C_VEL
LIN {X 0,Y 271.899,Z 685.43,A -85,B 0,C 180,E1 -18660.911,E2 -18660.911} C_VEL
LIN {X 0,Y 273.395,Z 672.475,A -85,B 0,C 180,E1 -18661.744,E2 -18661.744} C_VEL
LIN {X 0,Y 274.242,Z 659.272,A -85,B 0,C 180,E1 -18662.292,E2 -18662.292} C_VEL
LIN {X 0,Y 276.449,Z 596.687,A -85,B 0,C 180,E1 -18663.899,E2 -18663.899} C_VEL
LIN {X 0,Y 268.602,Z 578.537,A -85,B 0,C 180,E1 -18665.513,E2 -18665.513} C_VEL
LIN {X 0,Y 260.687,Z 562.838,A -85,B 0,C 180,E1 -18667.188,E2 -18667.188} C_VEL
LIN {X 0,Y 256.896,Z 555.616,A -85,B 0,C 180,E1 -18668.063,E2 -18668.063} C_VEL
LIN {X 0,Y 256.134,Z 552.581,A -85,B 0,C 180,E1 -18669.661,E2 -18669.661} C_VEL
LIN {X 0,Y 256.103,Z 552.582,A -85,B 0,C 180,E1 -18673.317,E2 -18673.317} C_VEL
LIN {X 0,Y 256.111,Z 552.572,A -85,B 0,C 180,E1 -18677.808,E2 -18677.808} C_VEL
LIN {X 0,Y 256.098,Z 552.581,A -85,B 0,C 180,E1 -18680.862,E2 -18680.862} C_VEL
LIN {X 0,Y 256.119,Z 552.582,A -85,B 0,C 180,E1 -18684.812,E2 -18684.812} C_VEL
LIN {X 0,Y 256.089,Z 552.583,A -85,B 0,C 180,E1 -18688.572,E2 -18688.572} C_VEL
LIN {X 0,Y 256.138,Z 552.579,A -85,B 0,C 180,E1 -18692.195,E2 -18692.195} C_VEL
LIN {X 0,Y 256.163,Z 552.576,A -85,B 0,C 180,E1 -18695.698,E2 -18695.698} C_VEL
LIN {X 0,Y 256.162,Z 552.575,A -85,B 0,C 180,E1 -18699.104,E2 -18699.104} C_VEL
LIN {X 0,Y 256.295,Z 552.558,A -85,B 0,C 180,E1 -18704.084,E2 -18704.084} C_VEL
LIN {X 0,Y 256.292,Z 552.558,A -85,B 0,C 180,E1 -18708.933,E2 -18708.933} C_VEL
LIN {X 0,Y 256.51,Z 552.522,A -85,B 0,C 180,E1 -18712.126,E2 -18712.126} C_VEL
LIN {X 0,Y 256.494,Z 552.526,A -85,B 0,C 180,E1 -18716.858,E2 -18716.858} C_VEL
LIN {X 0,Y 256.768,Z 552.499,A -85,B 0,C 180,E1 -18720,E2 -18720} C_VEL
LIN {X 0,Y 256.747,Z 552.5,A -85,B 0,C 180,E1 -18720.231,E2 -18720.231} C_VEL
LIN {X 0,Y 255.992,Z 552.595,A -85,B 0,C 180,E1 -18721.537,E2 -18721.537} C_VEL
LIN {X 0,Y 253.033,Z 552.964,A -85,B 0,C 180,E1 -18723.662,E2 -18723.662} C_VEL
LIN {X 0,Y 250.562,Z 553.273,A -85,B 0,C 180,E1 -18725.391,E2 -18725.391} C_VEL
LIN {X 0,Y 249.508,Z 553.403,A -85,B 0,C 180,E1 -18726.735,E2 -18726.735} C_VEL
LIN {X 0,Y 249.423,Z 553.408,A -85,B 0,C 180,E1 -18727.191,E2 -18727.191} C_VEL
LIN {X 0,Y 249.338,Z 553.421,A -85,B 0,C 180,E1 -18729.736,E2 -18729.736} C_VEL
LIN {X 0,Y 249.195,Z 553.437,A -85,B 0,C 180,E1 -18734.704,E2 -18734.704} C_VEL
LIN {X 0,Y 249.133,Z 553.443,A -85,B 0,C 180,E1 -18738.078,E2 -18738.078} C_VEL
LIN {X 0,Y 249.079,Z 553.457,A -85,B 0,C 180,E1 -18741.519,E2 -18741.519} C_VEL
LIN {X 0,Y 249.112,Z 553.453,A -85,B 0,C 180,E1 -18745.476,E2 -18745.476} C_VEL
LIN {X 0,Y 249.079,Z 553.459,A -85,B 0,C 180,E1 -18748.994,E2 -18748.994} C_VEL
LIN {X 0,Y 249.032,Z 553.463,A -85,B 0,C 180,E1 -18752.426,E2 -18752.426} C_VEL
LIN {X 0,Y 249.07,Z 553.459,A -85,B 0,C 180,E1 -18756.338,E2 -18756.338} C_VEL
LIN {X 0,Y 249.041,Z 553.466,A -85,B 0,C 180,E1 -18760.471,E2 -18760.471} C_VEL
LIN {X 0,Y 249.008,Z 553.471,A -85,B 0,C 180,E1 -18764.878,E2 -18764.878} C_VEL
LIN {X 0,Y 249.039,Z 553.642,A -85,B 0,C 180,E1 -18768.997,E2 -18768.997} C_VEL
LIN {X 0,Y 251.009,Z 560.901,A -85,B 0,C 180,E1 -18772.486,E2 -18772.486} C_VEL
LIN {X 0,Y 252.518,Z 567.177,A -85,B 0,C 180,E1 -18775.29,E2 -18775.29} C_VEL
LIN {X 0,Y 254.567,Z 571.406,A -85,B 0,C 180,E1 -18775.773,E2 -18775.773} C_VEL
LIN {X 0,Y 262.252,Z 587.502,A -85,B 0,C 180,E1 -18777.5,E2 -18777.5} C_VEL
LIN {X 0,Y 266.446,Z 597.779,A -85,B 0,C 180,E1 -18778.434,E2 -18778.434} C_VEL
LIN {X 0,Y 269.659,Z 618.093,A -85,B 0,C 180,E1 -18779.507,E2 -18779.507} C_VEL
LIN {X 0,Y 267.473,Z 676.512,A -85,B 0,C 180,E1 -18781.071,E2 -18781.071} C_VEL
LIN {X 0,Y 266.24,Z 690.322,A -85,B 0,C 180,E1 -18781.739,E2 -18781.739} C_VEL
LIN {X 0,Y 264.53,Z 702.618,A -85,B 0,C 180,E1 -18782.616,E2 -18782.616} C_VEL
LIN {X 0,Y 262.572,Z 714.422,A -85,B 0,C 180,E1 -18783.792,E2 -18783.792} C_VEL
LIN {X 0,Y 260.218,Z 725.79,A -85,B 0,C 180,E1 -18785.253,E2 -18785.253} C_VEL
LIN {X 0,Y 257.799,Z 736.051,A -85,B 0,C 180,E1 -18786.929,E2 -18786.929} C_VEL
LIN {X 0,Y 255.642,Z 744.451,A -85,B 0,C 180,E1 -18788.638,E2 -18788.638} C_VEL
LIN {X 0,Y 253.64,Z 752.213,A -85,B 0,C 180,E1 -18790.58,E2 -18790.58} C_VEL
LIN {X 0,Y 251.609,Z 759.811,A -85,B 0,C 180,E1 -18792.945,E2 -18792.945} C_VEL
LIN {X 0,Y 249.837,Z 765.936,A -85,B 0,C 180,E1 -18795.335,E2 -18795.335} C_VEL
LIN {X 0,Y 248.572,Z 770.807,A -85,B 0,C 180,E1 -18797.758,E2 -18797.758} C_VEL
LIN {X 0,Y 247.697,Z 774.566,A -85,B 0,C 180,E1 -18800.198,E2 -18800.198} C_VEL
LIN {X 0,Y 247.283,Z 776.512,A -85,B 0,C 180,E1 -18801.831,E2 -18801.831} C_VEL
LIN {X 0,Y 247.013,Z 778.043,A -85,B 0,C 180,E1 -18803.465,E2 -18803.465} C_VEL
LIN {X 0,Y 246.864,Z 779.816,A -85,B 0,C 180,E1 -18806.736,E2 -18806.736} C_VEL
LIN {X 0,Y 246.928,Z 780.123,A -85,B 0,C 180,E1 -18808.369,E2 -18808.369} C_VEL
LIN {X 0,Y 246.985,Z 780.04,A -85,B 0,C 180,E1 -18810,E2 -18810} C_VEL
LIN {X 0,Y 246.931,Z 779.52,A -85,B 0,C 180,E1 -18811.631,E2 -18811.631} C_VEL
LIN {X 0,Y 246.883,Z 778.596,A -85,B 0,C 180,E1 -18813.264,E2 -18813.264} C_VEL
LIN {X 0,Y 246.913,Z 777.202,A -85,B 0,C 180,E1 -18814.981,E2 -18814.981} C_VEL
LIN {X 0,Y 247.112,Z 774.475,A -85,B 0,C 180,E1 -18817.353,E2 -18817.353} C_VEL
LIN {X 0,Y 247.596,Z 770.642,A -85,B 0,C 180,E1 -18819.806,E2 -18819.806} C_VEL
LIN {X 0,Y 248.358,Z 765.674,A -85,B 0,C 180,E1 -18822.253,E2 -18822.253} C_VEL
LIN {X 0,Y 249.586,Z 759.427,A -85,B 0,C 180,E1 -18824.68,E2 -18824.68} C_VEL
LIN {X 0,Y 251.2,Z 751.624,A -85,B 0,C 180,E1 -18827.083,E2 -18827.083} C_VEL
LIN {X 0,Y 252.907,Z 742.899,A -85,B 0,C 180,E1 -18829.231,E2 -18829.231} C_VEL
LIN {X 0,Y 254.766,Z 732.813,A -85,B 0,C 180,E1 -18831.227,E2 -18831.227} C_VEL
LIN {X 0,Y 256.772,Z 721.671,A -85,B 0,C 180,E1 -18832.956,E2 -18832.956} C_VEL
LIN {X 0,Y 258.513,Z 710.741,A -85,B 0,C 180,E1 -18834.279,E2 -18834.279} C_VEL
LIN {X 0,Y 260.179,Z 698.67,A -85,B 0,C 180,E1 -18835.392,E2 -18835.392} C_VEL
LIN {X 0,Y 261.441,Z 686.286,A -85,B 0,C 180,E1 -18836.222,E2 -18836.222} C_VEL
